   statRcvBuffer[1317] := ' ';
   statRcvBuffer[1318] := ' ';
   statRcvBuffer[1319] := ' ';
   statRcvBuffer[1320] := ' ';
   statRcvBuffer[1321] := ' ';
   statRcvBuffer[1322] := ' ';
   statRcvBuffer[1323] := ' ';
   statRcvBuffer[1324] := ' ';
   statRcvBuffer[1325] := ' ';
   statRcvBuffer[1326] := ' ';
   statRcvBuffer[1327] := ' ';
   statRcvBuffer[1328] := ' ';
   statRcvBuffer[1329] := ' ';
   statRcvBuffer[1330] := ' ';
   statRcvBuffer[1331] := ' ';
   statRcvBuffer[1332] := ' ';
   statRcvBuffer[1333] := ' ';
   statRcvBuffer[1334] := ' ';
   statRcvBuffer[1335] := ' ';
   statRcvBuffer[1336] := ' ';
   statRcvBuffer[1337] := ' ';
   statRcvBuffer[1338] := ' ';
   statRcvBuffer[1339] := ' ';
   statRcvBuffer[1340] := ' ';
   statRcvBuffer[1341] := ' ';
   statRcvBuffer[1342] := ' ';
   statRcvBuffer[1343] := ' ';
   statRcvBuffer[1344] := ' ';
   statRcvBuffer[1345] := ' ';
   statRcvBuffer[1346] := ' ';
   statRcvBuffer[1347] := ' ';
   statRcvBuffer[1348] := ' ';
   statRcvBuffer[1349] := ' ';
   statRcvBuffer[1350] := ' ';
   statRcvBuffer[1351] := ' ';
   statRcvBuffer[1352] := ' ';
   statRcvBuffer[1353] := ' ';
   statRcvBuffer[1354] := ' ';
   statRcvBuffer[1355] := ' ';
   statRcvBuffer[1356] := ' ';
   statRcvBuffer[1357] := ' ';
   statRcvBuffer[1358] := ' ';
   statRcvBuffer[1359] := ' ';
   statRcvBuffer[1360] := ' ';
   statRcvBuffer[1361] := ' ';
   statRcvBuffer[1362] := ' ';
   statRcvBuffer[1363] := ' ';
   statRcvBuffer[1364] := ' ';
   statRcvBuffer[1365] := ' ';
   statRcvBuffer[1366] := ' ';
   statRcvBuffer[1367] := ' ';
   statRcvBuffer[1368] := ' ';
   statRcvBuffer[1369] := ' ';
   statRcvBuffer[1370] := ' ';
   statRcvBuffer[1371] := ' ';
   statRcvBuffer[1372] := ' ';
   statRcvBuffer[1373] := ' ';
   statRcvBuffer[1374] := ' ';
   statRcvBuffer[1375] := ' ';
   statRcvBuffer[1376] := ' ';
   statRcvBuffer[1377] := ' ';
   statRcvBuffer[1378] := ' ';
   statRcvBuffer[1379] := ' ';
   statRcvBuffer[1380] := ' ';
   statRcvBuffer[1381] := ' ';
   statRcvBuffer[1382] := ' ';
   statRcvBuffer[1383] := ' ';
   statRcvBuffer[1384] := ' ';
   statRcvBuffer[1385] := ' ';
   statRcvBuffer[1386] := ' ';
   statRcvBuffer[1387] := ' ';
   statRcvBuffer[1388] := ' ';
   statRcvBuffer[1389] := ' ';
   statRcvBuffer[1390] := ' ';
   statRcvBuffer[1391] := ' ';
   statRcvBuffer[1392] := ' ';
   statRcvBuffer[1393] := ' ';
   statRcvBuffer[1394] := ' ';
   statRcvBuffer[1395] := ' ';
   statRcvBuffer[1396] := ' ';
   statRcvBuffer[1397] := ' ';
   statRcvBuffer[1398] := ' ';
   statRcvBuffer[1399] := ' ';
   statRcvBuffer[1400] := ' ';
   statRcvBuffer[1401] := ' ';
   statRcvBuffer[1402] := ' ';
   statRcvBuffer[1403] := ' ';
   statRcvBuffer[1404] := ' ';
   statRcvBuffer[1405] := ' ';
   statRcvBuffer[1406] := ' ';
   statRcvBuffer[1407] := ' ';
   statRcvBuffer[1408] := ' ';
   statRcvBuffer[1409] := ' ';
   statRcvBuffer[1410] := ' ';
   statRcvBuffer[1411] := ' ';
   statRcvBuffer[1412] := ' ';
   statRcvBuffer[1413] := ' ';
   statRcvBuffer[1414] := ' ';
   statRcvBuffer[1415] := ' ';
   statRcvBuffer[1416] := ' ';
   statRcvBuffer[1417] := ' ';
   statRcvBuffer[1418] := ' ';
   statRcvBuffer[1419] := ' ';
   statRcvBuffer[1420] := ' ';
   statRcvBuffer[1421] := ' ';
   statRcvBuffer[1422] := ' ';
   statRcvBuffer[1423] := ' ';
   statRcvBuffer[1424] := ' ';
   statRcvBuffer[1425] := ' ';
   statRcvBuffer[1426] := ' ';
   statRcvBuffer[1427] := ' ';
   statRcvBuffer[1428] := ' ';
   statRcvBuffer[1429] := ' ';
   statRcvBuffer[1430] := ' ';
   statRcvBuffer[1431] := ' ';
   statRcvBuffer[1432] := ' ';
   statRcvBuffer[1433] := ' ';
   statRcvBuffer[1434] := ' ';
   statRcvBuffer[1435] := ' ';
   statRcvBuffer[1436] := ' ';
   statRcvBuffer[1437] := ' ';
   statRcvBuffer[1438] := ' ';
   statRcvBuffer[1439] := ' ';
   statRcvBuffer[1440] := ' ';
   statRcvBuffer[1441] := ' ';
   statRcvBuffer[1442] := ' ';
   statRcvBuffer[1443] := ' ';
   statRcvBuffer[1444] := ' ';
   statRcvBuffer[1445] := ' ';
   statRcvBuffer[1446] := ' ';
   statRcvBuffer[1447] := ' ';
   statRcvBuffer[1448] := ' ';
   statRcvBuffer[1449] := ' ';
   statRcvBuffer[1450] := ' ';
   statRcvBuffer[1451] := ' ';
   statRcvBuffer[1452] := ' ';
   statRcvBuffer[1453] := ' ';
   statRcvBuffer[1454] := ' ';
   statRcvBuffer[1455] := ' ';
   statRcvBuffer[1456] := ' ';
   statRcvBuffer[1457] := ' ';
   statRcvBuffer[1458] := ' ';
   statRcvBuffer[1459] := ' ';
   statSizeRcvArray := 101;
   statDataIsString := TRUE;
END_DATA_BLOCK

DATA_BLOCK "LHTTP_parameters"   // DB3
{ S7_Optimized_Access := 'TRUE' }
VERSION : 0.1
   VAR
      hwID : Hw_Any := 0;
      connID : Conn_Ouc := 16#0001;
      url : String := '192.168.0.56:55555/resource';
      contentType : String := 'application/json';
      Head : String := 'Authorization: Basic dGVzdDEyMzQ1OnRlc3QxMjM0NQ==$00';
      HeaderData : Array[0..255] of Char;
      responseData : Array[0..100] of Char;
   END_VAR
BEGIN
   responseData[100] := ' ';
   responseData[99] := ' ';
   responseData[98] := ' ';
   responseData[97] := ' ';
   responseData[96] := ' ';
   responseData[95] := ' ';
   responseData[94] := ' ';
   responseData[93] := ' ';
   responseData[92] := ' ';
   responseData[91] := ' ';
   responseData[90] := ' ';
   responseData[89] := ' ';
   responseData[88] := ' ';
   responseData[87] := ' ';
   responseData[86] := ' ';
   responseData[85] := ' ';
   responseData[84] := ' ';
   responseData[83] := ' ';
   responseData[82] := ' ';
   responseData[81] := ' ';
   responseData[80] := ' ';
   responseData[79] := '}';
   responseData[78] := '"';
   responseData[77] := 'e';
   responseData[76] := 'c';
   responseData[75] := 'r';
   responseData[74] := 'u';
   responseData[73] := 'o';
   responseData[72] := 's';
   responseData[71] := 'e';
   responseData[70] := 'r';
   responseData[69] := ' ';
   responseData[68] := 'e';
   responseData[67] := 'l';
   responseData[66] := 'p';
   responseData[65] := 'm';
   responseData[64] := 'a';
   responseData[63] := 'x';
   responseData[62] := 'e';
   responseData[61] := ' ';
   responseData[60] := 'n';
   responseData[59] := 'a';
   responseData[58] := ' ';
   responseData[57] := 's';
   responseData[56] := 'i';
   responseData[55] := ' ';
   responseData[54] := 's';
   responseData[53] := 'i';
   responseData[52] := 'h';
   responseData[51] := 'T';
   responseData[50] := '"';
   responseData[49] := ':';
   responseData[48] := '"';
   responseData[47] := 'n';
   responseData[46] := 'o';
   responseData[45] := 'i';
   responseData[44] := 't';
   responseData[43] := 'p';
   responseData[42] := 'i';
   responseData[41] := 'r';
   responseData[40] := 'c';
   responseData[39] := 's';
   responseData[38] := 'e';
   responseData[37] := 'd';
   responseData[36] := '"';
   responseData[35] := ',';
   responseData[34] := '"';
   responseData[33] := 'e';
   responseData[32] := 'c';
   responseData[31] := 'r';
   responseData[30] := 'u';
   responseData[29] := 'o';
   responseData[28] := 's';
   responseData[27] := 'e';
   responseData[26] := 'r';
   responseData[25] := ' ';
   responseData[24] := 'e';
   responseData[23] := 'l';
   responseData[22] := 'p';
   responseData[21] := 'm';
   responseData[20] := 'a';
   responseData[19] := 'x';
   responseData[18] := 'e';
   responseData[17] := '"';
   responseData[16] := ':';
   responseData[15] := '"';
   responseData[14] := 'e';
   responseData[13] := 'm';
   responseData[12] := 'a';
   responseData[11] := 'n';
   responseData[10] := '"';
   responseData[9] := ',';
   responseData[8] := '"';
   responseData[7] := '1';
   responseData[6] := '"';
   responseData[5] := ':';
   responseData[4] := '"';
   responseData[3] := 'd';
   responseData[2] := 'i';
   responseData[1] := '"';
   responseData[0] := '{';
   HeaderData[0] := 'A';
   HeaderData[1] := 'u';
   HeaderData[2] := 't';
   HeaderData[3] := 'h';
   HeaderData[4] := 'o';
   HeaderData[5] := 'r';
   HeaderData[6] := 'i';
   HeaderData[7] := 'z';
   HeaderData[8] := 'a';
   HeaderData[9] := 't';
   HeaderData[10] := 'i';
   HeaderData[11] := 'o';
   HeaderData[12] := 'n';
   HeaderData[13] := ':';
   HeaderData[14] := ' ';
   HeaderData[15] := 'B';
   HeaderData[16] := 'a';
   HeaderData[17] := 's';
   HeaderData[18] := 'i';
   HeaderData[19] := 'c';
   HeaderData[20] := ' ';
   HeaderData[21] := 'd';
   HeaderData[22] := 'G';
   HeaderData[23] := 'V';
   HeaderData[24] := 'z';
   HeaderData[25] := 'd';
   HeaderData[26] := 'D';
   HeaderData[27] := 'E';
   HeaderData[28] := 'y';
   HeaderData[29] := 'M';
   HeaderData[30] := 'z';
   HeaderData[31] := 'Q';
   HeaderData[32] := '1';
   HeaderData[33] := 'O';
   HeaderData[34] := 'n';
   HeaderData[35] := 'R';
   HeaderData[36] := 'l';
   HeaderData[37] := 'c';
   HeaderData[38] := '3';
   HeaderData[39] := 'Q';
   HeaderData[40] := 'x';
   HeaderData[41] := 'M';
   HeaderData[42] := 'j';
   HeaderData[43] := 'M';
   HeaderData[44] := '0';
   HeaderData[45] := 'N';
   HeaderData[46] := 'Q';
   HeaderData[47] := '=';
   HeaderData[48] := '=';
   HeaderData[49] := '$00';
   HeaderData[50] := ' ';
   HeaderData[51] := ' ';
   HeaderData[52] := ' ';
   HeaderData[53] := ' ';
   HeaderData[54] := ' ';
   HeaderData[55] := ' ';
   HeaderData[56] := ' ';
   HeaderData[57] := ' ';
   HeaderData[58] := ' ';
   HeaderData[59] := ' ';
   HeaderData[60] := ' ';
   HeaderData[61] := ' ';
   HeaderData[62] := ' ';
   HeaderData[63] := ' ';
   HeaderData[64] := ' ';
   HeaderData[65] := ' ';
   HeaderData[66] := ' ';
   HeaderData[67] := ' ';
   HeaderData[68] := ' ';
   HeaderData[69] := ' ';
   HeaderData[70] := ' ';
   HeaderData[71] := ' ';
   HeaderData[72] := ' ';
   HeaderData[73] := ' ';
   HeaderData[74] := ' ';
   HeaderData[75] := ' ';
   HeaderData[76] := ' ';
   HeaderData[77] := ' ';
   HeaderData[78] := ' ';
   HeaderData[79] := ' ';
   HeaderData[80] := ' ';
   HeaderData[81] := ' ';
   HeaderData[82] := ' ';
   HeaderData[83] := ' ';
   HeaderData[84] := ' ';
   HeaderData[85] := ' ';
   HeaderData[86] := ' ';
   HeaderData[87] := ' ';
   HeaderData[88] := ' ';
   HeaderData[89] := ' ';
   HeaderData[90] := ' ';
   HeaderData[91] := ' ';
   HeaderData[92] := ' ';
   HeaderData[93] := ' ';
   HeaderData[94] := ' ';
   HeaderData[95] := ' ';
   HeaderData[96] := ' ';
   HeaderData[97] := ' ';
   HeaderData[98] := ' ';
   HeaderData[99] := ' ';
   HeaderData[100] := ' ';
   HeaderData[101] := ' ';
   HeaderData[102] := ' ';
   HeaderData[103] := ' ';
   HeaderData[104] := ' ';
   HeaderData[105] := ' ';
   HeaderData[106] := ' ';
   HeaderData[107] := ' ';
   HeaderData[108] := ' ';
   HeaderData[109] := ' ';
   HeaderData[110] := ' ';
   HeaderData[111] := ' ';
   HeaderData[112] := ' ';
   HeaderData[113] := ' ';
   HeaderData[114] := ' ';
   HeaderData[115] := ' ';
   HeaderData[116] := ' ';
   HeaderData[117] := ' ';
   HeaderData[118] := ' ';
   HeaderData[119] := ' ';
   HeaderData[120] := ' ';
   HeaderData[121] := ' ';
   HeaderData[122] := ' ';
   HeaderData[123] := ' ';
   HeaderData[124] := ' ';
   HeaderData[125] := ' ';
   HeaderData[126] := ' ';
   HeaderData[127] := ' ';
   HeaderData[128] := ' ';
   HeaderData[129] := ' ';
   HeaderData[130] := ' ';
   HeaderData[131] := ' ';
   HeaderData[132] := ' ';
   HeaderData[133] := ' ';
   HeaderData[134] := ' ';
   HeaderData[135] := ' ';
   HeaderData[136] := ' ';
   HeaderData[137] := ' ';
   HeaderData[138] := ' ';
   HeaderData[139] := ' ';
   HeaderData[140] := ' ';
   HeaderData[141] := ' ';
   HeaderData[142] := ' ';
   HeaderData[143] := ' ';
   HeaderData[144] := ' ';
   HeaderData[145] := ' ';
   HeaderData[146] := ' ';
   HeaderData[147] := ' ';
   HeaderData[148] := ' ';
   HeaderData[149] := ' ';
   HeaderData[150] := ' ';
   HeaderData[151] := ' ';
   HeaderData[152] := ' ';
   HeaderData[153] := ' ';
   HeaderData[154] := ' ';
   HeaderData[155] := ' ';
   HeaderData[156] := ' ';
   HeaderData[157] := ' ';
   HeaderData[158] := ' ';
   HeaderData[159] := ' ';
   HeaderData[160] := ' ';
   HeaderData[161] := ' ';
   HeaderData[162] := ' ';
   HeaderData[163] := ' ';
   HeaderData[164] := ' ';
   HeaderData[165] := ' ';
   HeaderData[166] := ' ';
   HeaderData[167] := ' ';
   HeaderData[168] := ' ';
   HeaderData[169] := ' ';
   HeaderData[170] := ' ';
   HeaderData[171] := ' ';
   HeaderData[172] := ' ';
   HeaderData[173] := ' ';
   HeaderData[174] := ' ';
   HeaderData[175] := ' ';
   HeaderData[176] := ' ';
   HeaderData[177] := ' ';
   HeaderData[178] := ' ';
   HeaderData[179] := ' ';
   HeaderData[180] := ' ';
   HeaderData[181] := ' ';
   HeaderData[182] := ' ';
   HeaderData[183] := ' ';
   HeaderData[184] := ' ';
   HeaderData[185] := ' ';
   HeaderData[186] := ' ';
   HeaderData[187] := ' ';
   HeaderData[188] := ' ';
   HeaderData[189] := ' ';
   HeaderData[190] := ' ';
   HeaderData[191] := ' ';
   HeaderData[192] := ' ';
   HeaderData[193] := ' ';
   HeaderData[194] := ' ';
   HeaderData[195] := ' ';
   HeaderData[196] := ' ';
   HeaderData[197] := ' ';
   HeaderData[198] := ' ';
   HeaderData[199] := ' ';
   HeaderData[200] := ' ';
   HeaderData[201] := ' ';
   HeaderData[202] := ' ';
   HeaderData[203] := ' ';
   HeaderData[204] := ' ';
   HeaderData[205] := ' ';
   HeaderData[206] := ' ';
   HeaderData[207] := ' ';
   HeaderData[208] := ' ';
   HeaderData[209] := ' ';
   HeaderData[210] := ' ';
   HeaderData[211] := ' ';
   HeaderData[212] := ' ';
   HeaderData[213] := ' ';
   HeaderData[214] := ' ';
   HeaderData[215] := ' ';
   HeaderData[216] := ' ';
   HeaderData[217] := ' ';
   HeaderData[218] := ' ';
   HeaderData[219] := ' ';
   HeaderData[220] := ' ';
   HeaderData[221] := ' ';
   HeaderData[222] := ' ';
   HeaderData[223] := ' ';
   HeaderData[224] := ' ';
   HeaderData[225] := ' ';
   HeaderData[226] := ' ';
   HeaderData[227] := ' ';
   HeaderData[228] := ' ';
   HeaderData[229] := ' ';
   HeaderData[230] := ' ';
   HeaderData[231] := ' ';
   HeaderData[232] := ' ';
   HeaderData[233] := ' ';
   HeaderData[234] := ' ';
   HeaderData[235] := ' ';
   HeaderData[236] := ' ';
   HeaderData[237] := ' ';
   HeaderData[238] := ' ';
   HeaderData[239] := ' ';
   HeaderData[240] := ' ';
   HeaderData[241] := ' ';
   HeaderData[242] := ' ';
   HeaderData[243] := ' ';
   HeaderData[244] := ' ';
   HeaderData[245] := ' ';
   HeaderData[246] := ' ';
   HeaderData[247] := ' ';
   HeaderData[248] := ' ';
   HeaderData[249] := ' ';
   HeaderData[250] := ' ';
   HeaderData[251] := ' ';
   HeaderData[252] := ' ';
   HeaderData[253] := ' ';
   HeaderData[254] := ' ';
   HeaderData[255] := ' ';
END_DATA_BLOCK

DATA_BLOCK "LHTTP_control"   // DB5
{ S7_Optimized_Access := 'TRUE' }
VERSION : 0.1
   VAR
      PUT_POST : Bool;
      GET : Bool;
      ExtractedDataName : String;
      ExtractedDataDescription : String;
      ExtractedDataMessage : String;
      RequestPayload : String := '{"id":"1","name":"example resource","description":"This is an example resource"}';
      geturl : String := '192.168.0.56:55555/resource/1';
      PostOrPut : USInt := 0;   // 0=post , 1=put
   END_VAR
BEGIN
END_DATA_BLOCK

// folder: (top level)

ORGANIZATION_BLOCK "Main"   // OB1, LAD, ProgramCycle
TITLE = "Main Program Sweep (Cycle)"
{ S7_Optimized_Access := 'TRUE' }
VERSION : 0.1
   VAR_INPUT
      Initial_Call : Bool;   // Initial call of this OB
      Remanence : Bool;   // =True, if remanent data are available
   END_VAR
BEGIN

REGION Network 1
   // Download password 1234
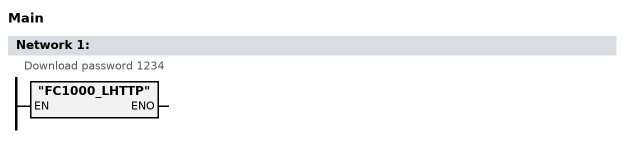
   RUNG wire#powerrail
      "FC1000_LHTTP"()
   END_RUNG
   // the same network as SCL:
   "FC1000_LHTTP"();
END_REGION
END_ORGANIZATION_BLOCK

// folder: 1000_HTTP

FUNCTION "FC1000_LHTTP" : Void   // FC1000, FBD
{ S7_Optimized_Access := 'TRUE' }
VERSION : 0.1
BEGIN

REGION Network 1: Header Data Additions - Convert String to Chars
   // Header fields are separated by an end-ofline ("$R$L"). The end of the user-defined header fields is signaled to the FB with the character 
   // "$00"
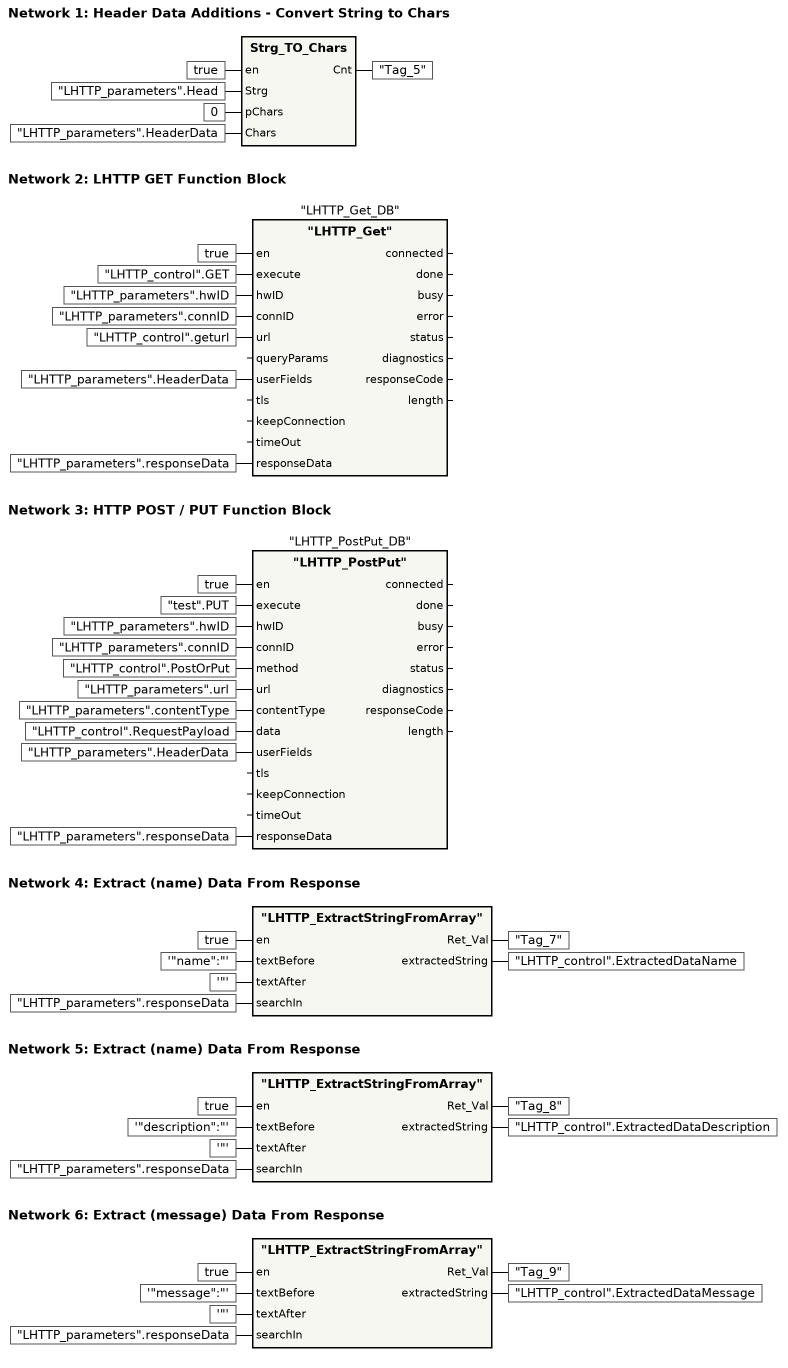
   // no SCL statement known for Strg_TO_Chars: written as a call
   IF true THEN
       Strg_TO_Chars(Strg := "LHTTP_parameters".Head,
                     pChars := 0,
                     Chars := "LHTTP_parameters".HeaderData,
                     Cnt => "Tag_5");
   END_IF;
END_REGION

REGION Network 2: LHTTP GET Function Block
   IF true THEN
       "LHTTP_Get_DB"(execute := "LHTTP_control".GET,   // "LHTTP_Get"
                      hwID := "LHTTP_parameters".hwID,
                      connID := "LHTTP_parameters".connID,
                      url := "LHTTP_control".geturl,
                      userFields := "LHTTP_parameters".HeaderData,
                      responseData := "LHTTP_parameters".responseData);
   END_IF;
END_REGION

REGION Network 3: HTTP POST / PUT Function Block
   IF true THEN
       "LHTTP_PostPut_DB"(execute := "test".PUT,   // "LHTTP_PostPut"
                          hwID := "LHTTP_parameters".hwID,
                          connID := "LHTTP_parameters".connID,
                          method := "LHTTP_control".PostOrPut,
                          url := "LHTTP_parameters".url,
                          contentType := "LHTTP_parameters".contentType,
                          data := "LHTTP_control".RequestPayload,
                          userFields := "LHTTP_parameters".HeaderData,
                          responseData := "LHTTP_parameters".responseData);
   END_IF;
END_REGION

REGION Network 4: Extract (name) Data From Response
   IF true THEN
       "Tag_7" := "LHTTP_ExtractStringFromArray"(textBefore := '"name":"',
                               textAfter := '"',
                               searchIn := "LHTTP_parameters".responseData,
                               extractedString => "LHTTP_control".ExtractedDataName);
   END_IF;
END_REGION

REGION Network 5: Extract (name) Data From Response
   IF true THEN
       "Tag_8" := "LHTTP_ExtractStringFromArray"(textBefore := '"description":"',
                               textAfter := '"',
                               searchIn := "LHTTP_parameters".responseData,
                               extractedString => "LHTTP_control".ExtractedDataDescription);
   END_IF;
END_REGION

REGION Network 6: Extract (message) Data From Response
   IF true THEN
       "Tag_9" := "LHTTP_ExtractStringFromArray"(textBefore := '"message":"',
                               textAfter := '"',
                               searchIn := "LHTTP_parameters".responseData,
                               extractedString => "LHTTP_control".ExtractedDataMessage);
   END_IF;
END_REGION
END_FUNCTION

// folder: 1000_HTTP/LHTTP

FUNCTION_BLOCK "LHTTP_Get"   // FB8, SCL
TITLE = LHTTP_Get
{ S7_Optimized_Access := 'TRUE' }
AUTHOR : Siemens Industry Online Support
FAMILY : LHTTP
VERSION : 2.1
// Implements the HTTP GET method
   VAR_INPUT
      execute : Bool;   // Send HTTP request
      hwID : Hw_Any;   // Hardware ID of Ethernet interface
      connID : Conn_Ouc := 1;   // Unique connection ID
      url : String;   // URL, i.e. "http://www.siemens.com/simatic"
      queryParams : String;   // Additional query parameters if "url" is not long enough, i.e. "lang=en&q=simatic"; "?" or "&" is inserted automatically in between "url" and "queryParameters". / Optional query parameters that are appended to URL, i.e. "lang=en&q=simatic"
      userFields : Array[0..#UPPER_USER_FIELDS] of Char;   // Additional user-defined header fields
      tls : "LHTTP_typeTLS";   // TLS certificates for secure connections (HTTPS), leave open for non-secure connections (HTTP)
      keepConnection : Bool;   // Keep connection established after execution of request
      timeOut : Time := T#10s;   // Time to wait for response from server
   END_VAR
   VAR_OUTPUT
      connected : Bool;   // Connection to web server is established
      done : Bool;   // HTTP request finished
      busy : Bool;   // Function is busy
      error : Bool;   // An error occured
      status : Word := 16#7000;   // Specifies the error
      diagnostics : "typeDiagnostics";   // Diagnostics information of FB
      responseCode : UInt;   // HTTP response code
      length : UDInt;   // Length of received data
   END_VAR
   VAR_IN_OUT
      responseData : Array[*] of Char;   // Data received from HTTP server
   END_VAR
   VAR
      instTSendC : TSEND_C;   // Instance of TSEND_C
      instTRcv : TRCV;   // Instance of TRCV
      instTimeout : TON_TIME;   // Time-out
      statConnected : Bool;   // Static value for output 'connected'
      statDone : Bool;   // Static value for output 'done'
      statBusy : Bool;   // Static value for output 'busy'
      statError : Bool;   // Static value for output 'error'
      statStatus : Word := 16#7000;   // Static value for output 'status'
      statResponseCode : UInt;   // Static value for output 'responseCode'
      statLength : UDInt;   // Static value for output 'length'
      statFBState : USInt := 0;   // Current state in state machine
      statSubfunctionStatus : DWord;   // Status or return value of called FBs, FCs and system blocks
      statEmptyDiagnostics : "typeDiagnostics";   // Empty diagnostics information (for initialization purposes only)
      statParam : Struct   // Connection parameters
         isQDN : Bool;
         paramQDN : TCON_QDN_SEC;   // Connection parameters in form of QDN
         paramIP : TCON_IP_V4_SEC;   // Connection parameters in form of IP address
      END_STRUCT;
      statHost : String;   // Host part of URL
      statRequest : Struct   // GET request
         chars : Array[0..#UPPER_REQUEST_ARRAY] of Char;   // GET request (max. length: url (254) + data (254) + header (94)
         length : UInt;   // Length of GET request
      END_STRUCT;
      statSend : Struct   // Parameters for instruction TSend_C
         connect : Bool;   // Establish and keep connection
         req : Bool;   // Send data
      END_STRUCT;
      statEncoding : String;   // Transfer encoding of response from HTTP server
      statContentLength : UInt;   // Content length as specified in header of response
      statChunkLen : UDInt;   // Remaining length of current chunk
      statRcvdLen : UDInt;   // Sum length of received data
      statTimeoutIn : Bool;   // Timeout
      statRcvBuffer : Array[0..#UPPER_TCP_FRAME] of Char;   // Temporary receive buffer
      statSizeRcvArray : UDInt;   // Size of receive buffer at parameter "responseData"
      statExecuteOld : Bool;   // Last cycle's value of input "execute"
   END_VAR
   VAR_TEMP
      tempUrl : String;   // Copy of URL
      tempQuery : String;   // Query part of URL
      tempIndex : DInt;   // Index for for loops
      tempPos : Int;   // General tag for positions
      tempLen : UInt;   // General tag for lengths
      tempRet : Word;   // General tag for return values
      tempString : String;   // General tag for strings
      tempExitLoop : Bool;   // Condition to exit REPEAT loop around state machine
      tempChunk : Struct   // Temporary tags for chunked encoding
         posData : UInt;   // Start position of data in current packet
         lenData : UInt;   // Length of data in current packet
         exitLoop : Bool;   // Condition to exit loop
      END_STRUCT;
   END_VAR
   VAR CONSTANT
      UPPER_REQUEST_ARRAY : UInt := 1459;   // Upper limit of request array
      UPPER_TCP_FRAME : UInt := 1459;   // Upper limit of a TCP/IP frame
      UPPER_USER_FIELDS : USInt := 255;   // Upper limit of userFields
      PORT_UNSECURE : UInt := 80;   // Port for unsecure HTTP connection
      PORT_SECURE : UInt := 443;   // Port for secure HTTP connection
      POS_RESPONSE_CODE : USInt := 9;   // Position of HTTP response code in response message
      STATUS_DONE : Word := 16#0000;   // Job finished without errors
      STATUS_DISCONNECTED : Word := 16#0003;   // Communication connection closed
      STATUS_IDLE : Word := 16#7000;   // No job
      STATUS_FIRST_CALL : Word := 16#7001;   // First call after incoming new job (rising edge 'execute')
      STATUS_CONNECTING : Word := 16#7002;   // Connection is currently being established
      STATUS_DISCONNECTING : Word := 16#7003;   // Communication connection is being terminated
      STATUS_MONITORING : Word := 16#7004;   // Communication connection has been established and is being monitored. No send job execution active
      STATUS_SENT : Word := 16#7005;   // Request sent, waiting for response
      SUB_STATUS_NO_ERROR : DWord := 16#0000_0000;   // No error occured in subfunction call
      ERR_BOUND_NOT_ZERO : Word := 16#8201;   // Lower bound of receive buffer is not 0
      ERR_INVALID_URL : Word := 16#8202;   // Invalid URL
      ERR_DIFFERENT_HOST : Word := 16#8203;   // Trying to use existing connection with different host
      ERR_END_USER_FIELDS : Word := 16#8206;   // End of user-defined header fields could not be found
      ERR_REQUEST_SIZE : Word := 16#8210;   // Request array is too small for specified parameters
      ERR_RESPONSE_SIZE : Word := 16#8220;   // Receive buffer at parameter "responseData" too small
      ERR_CONN_LOST : Word := 16#8400;   // Offset for lost connection
      ERR_FORWARDING : Word := 16#8403;   // Server responded with forwarding message. Forwarding is not supported, see "diagnostics"
      ERR_WEBSERVER : Word := 16#8404;   // Webserver responded with error code, see "diagnostics"
      ERR_INVALID_HEADER : Word := 16#8405;   // Header of response is invalid
      ERR_TIMEOUT : Word := 16#8408;   // Time-out occurred
      ERR_UNDEFINED_STATE : Word := 16#8600;   // Error due to an undefined state in state machine
      ERR_TSENDC : Word := 16#8601;   // Error: TCON encountered an error, see "diagnostics"
      ERR_TRCV : Word := 16#8603;   // Error: TURCV encountered error, see "diagnostics"
      ERR_MOVE_USER_FIELDS : Word := 16#8612;   // Error in MOVE_BLK_VARIANT to copy user-defined header fields, see "diagnostics"
      ERR_ENCODING_UNKNOWN : Word := 16#8620;   // Transfer encoding of response could not be detected or is unsupported
      ERR_MOVE_IDENTITY : Word := 16#8630;   // Error in MOVE_BLK_VARIANT for transfer encoding 'identity', see "diagnostics"
      ERR_DECODING_FAILED : Word := 16#8640;   // Chunk encoded response could not be decoded
      ERR_MOVE_CHUNKED : Word := 16#8641;   // Error in MOVE_BLK_VARIANT for transfer encoding 'chunked', see "diagnostics"
      TSENDC_STATUS_CONNECTED : Word := 16#0001;   // TSEND_C: Communication connection established
      MOVE_STATUS_SIZE : Word := 16#8483;   // MOVE_BLK_VARIANT: DEST too small
      FB_STATE_NO_PROCESSING : USInt := 0;   // FB state: No processing
      FB_STATE_INIT : USInt := 1;   // FB state: initialization
      FB_STATE_REQUEST : USInt := 2;   // FB state: prepare request
      FB_STATE_SEND : USInt := 3;   // FB state: send request
      FB_STATE_RCV : USInt := 4;   // FB state: receive data
      FB_STATE_MON : USInt := 5;   // FB state: monitoring connection
      CRLF : String := '$R$L';   // Newline control character (carriage return, line feed)
      HEADER_END : String := '$R$L$R$L';   // End of HTTP header (two newline control characters)
      LEN_CRLF : UInt := 2;   // Length of CRLF
   END_VAR
   // statParam.paramIP.ConnPara.ActiveEstablished := true;
   // statParam.paramQDN.ConnPara.ActiveEstablished := true;
BEGIN
   REGION BLOCK INFO HEADER
     //===============================================================================
     // SIEMENS / (c)Copyright 2021
     //-------------------------------------------------------------------------------
     // Title:        LHTTP_Get
     // Function:     Implements the HTTP GET method
     // Library:      LHTTP
     // Author:       Siemens Industry Online Support
     // Tested with:  CPU 1516-3 PN/DP V2.9
     // Engineering:  TIA Portal V17
     // Restrictions: --
     // Requirements: S7-1200 with firmware V4.4 or higher
     //               S7-1500 with firmware V2.0 or higher
     //-------------------------------------------------------------------------------
     // Change log table:
     // Version  | Date       | Expert in charge       | Changes applied
     //----------|------------|------------------------|------------------------------
     // 02.01.00 | 2021-12-15 | Online Support         | Renamed parameter "data" to "queryParams"
     //-------------------------------------------------------------------------------
     // 02.00.04 | 2021-05-10 | Online Support         | Fixed issues with chunked encoding
     //          |            |                        | Allow chunk sizes > 65535 Bytes
     //          |            |                        | Made header evaluation case-insensitive
     //-------------------------------------------------------------------------------
     // 02.00.00 | 2020-12-16 | Online Support         | Added option to keep connection established
     //          |            |                        | Added parameter to add user-defined headers fields
     //          |            |                        | Changed to data type of "data" to Variant to allow larger data
     //          |            |                        | Removed "statusID" and added "diagnostics" instead, changed some error codes
     //-------------------------------------------------------------------------------
     // 01.00.00 | 2019-04-01 | Online Support         | First released version
     //===============================================================================
   END_REGION

   REGION INSTRUCTIONS
     IF (#statStatus <> #STATUS_IDLE) THEN // Only execute when FB is triggered to reduce system load
       // Connect and send
       IF #statParam.isQDN THEN // Call if host is a domain name
         #instTSendC(REQ     := #statSend.req,
                     CONT    := #statSend.connect,
                     LEN     := #statRequest.length,
                     CONNECT := #statParam.paramQDN,
                     DATA    := #statRequest.chars);
       ELSE // Call if host is an IP address
         #instTSendC(REQ     := #statSend.req,
                     CONT    := #statSend.connect,
                     LEN     := #statRequest.length,
                     CONNECT := #statParam.paramIP,
                     DATA    := #statRequest.chars);
       END_IF;

       // Receive
       #instTRcv(ID    := #statParam.paramQDN.ConnPara.ID,
                 EN_R  := #statFBState >= #FB_STATE_RCV,
                 LEN   := 0,
                 ADHOC := true,
                 DATA  := #statRcvBuffer);

       // Monitor time out
       #instTimeout(IN := #statTimeoutIn,
                    PT := #timeOut);

       IF #instTimeout.Q THEN
         #statStatus := #ERR_TIMEOUT;
       END_IF;
     END_IF;
   END_REGION

   REGION TRIGGERING
     IF (#execute = true AND #statExecuteOld = false) // Check if FB is triggered
       AND (#statStatus = #STATUS_IDLE OR #statStatus = #STATUS_MONITORING)
     THEN // First call; initialize FB
       // Copy URL
       #tempUrl := #url;

       #statBusy := true;
       #statStatus := #STATUS_FIRST_CALL;
       #statSubfunctionStatus := #SUB_STATUS_NO_ERROR;
       #diagnostics := #statEmptyDiagnostics;

       IF #statConnected = FALSE THEN // Connection is not yet established
         #statFBState := #FB_STATE_INIT;
       ELSE // Connection is already established, skip init
         #statFBState := #FB_STATE_REQUEST;
       END_IF;

     ELSIF (#statStatus = #STATUS_FIRST_CALL) THEN
       #statStatus := #STATUS_CONNECTING;
     END_IF;

     // Edge detection 'execute' input
     #statExecuteOld := #execute;
   END_REGION TRIGGERING

   IF (#statStatus = #STATUS_IDLE) THEN // Nothing to do -> End here to reduce "system load"
     RETURN;
   END_IF;

   REGION STATE_MACHINE
     // State machine is wrapped in REPEAT loop to make it possible to quickly exit state machine
     // in case of an error or to go through CASE multiple times within one cycle
     REPEAT
       #tempExitLoop := true; // Condition to exit loop is set per default

       CASE #statFBState OF // State machine of FB
         #FB_STATE_NO_PROCESSING: // No processing active
           ;

         #FB_STATE_INIT:
           REGION INIT
             // Get size of receive buffer
             IF LOWER_BOUND(ARR := #responseData, DIM := 1) <> 0 THEN
               #statStatus := #ERR_BOUND_NOT_ZERO;
               EXIT;
             ELSE
               #statSizeRcvArray := DINT_TO_UDINT(UPPER_BOUND(ARR := #responseData, DIM := 1)) + 1;
             END_IF;

             // Set connection parameters
             #statParam.paramQDN.ConnPara.InterfaceId := #hwID;
             #statParam.paramQDN.ConnPara.ID := #connID;
             #statParam.paramIP.ConnPara.InterfaceId := #hwID;
             #statParam.paramIP.ConnPara.ID := #connID;

             // Check if network protocol was specified to determine if connection should be secured
             #tempPos := FIND(IN1 := #tempUrl, IN2 := 'https://');
             IF #tempPos = 1 THEN // HTTPS
               #statParam.paramQDN.ActivateSecureConn := true;
               #statParam.paramQDN.ExtTLSCapabilities.%X0 := #tls.validateServerIdentity;
               #statParam.paramQDN.TLSServerCertRef := #tls.serverCert;
               #statParam.paramQDN.TLSClientCertRef := #tls.clientCert;
               #statParam.paramIP.ActivateSecureConn := true;
               #statParam.paramIP.ExtTLSCapabilities.%X0 := #tls.validateServerIdentity;
               #statParam.paramIP.TLSServerCertRef := #tls.serverCert;
               #statParam.paramIP.TLSClientCertRef := #tls.clientCert;
               // Delete network protocol from URL
               #tempUrl := DELETE(IN := #tempUrl, L := 8, P := 1);
             ELSE // HTTP
               #statParam.paramQDN.ActivateSecureConn := false;
               #statParam.paramIP.ActivateSecureConn := false;
               // Delete network protocol from URL if specified
               IF #tempUrl[5] = ':' THEN
                 #tempUrl := DELETE(IN := #tempUrl, L := 7, P := 1);
               END_IF;
             END_IF;

             // Determine if host is domain name or IP address
             #tempPos := CHAR_TO_INT(#tempUrl[1]);
             IF #tempPos >= CHAR_TO_INT('A') AND #tempPos <= CHAR_TO_INT('z') THEN // Host is a domain name
               #statParam.isQDN := true;
             ELSIF #tempPos >= CHAR_TO_INT('0') AND #tempPos <= CHAR_TO_INT('9') THEN // Host is an IP address
               #statParam.isQDN := false;
             ELSE // URL invalid
               #statStatus := #ERR_INVALID_URL;
               EXIT;
             END_IF;

             // Get host name and port
             #tempPos := FIND(IN1 := #tempUrl, IN2 := '/');
             IF #tempPos > 0 THEN // URL has a path after host name
               #statHost := LEFT(IN := #tempUrl, L := #tempPos - 1);
             ELSE
               #statHost := #tempUrl;
             END_IF;
             #tempPos := FIND(IN1 := #statHost, IN2 := ':');
             IF #tempPos > 0 THEN // Port specified in URL
               #statParam.paramQDN.ConnPara.RemotePort := STRING_TO_UINT(DELETE(IN := #statHost, L := #tempPos, P := 1));
               #statParam.paramIP.ConnPara.RemotePort := STRING_TO_UINT(DELETE(IN := #statHost, L := #tempPos, P := 1));
               #statHost := LEFT(IN := #statHost, L := #tempPos - 1);
             ELSE // No port specified in URL, set default port
               IF #statParam.paramQDN.ActivateSecureConn OR #statParam.paramIP.ActivateSecureConn THEN
                 #statParam.paramQDN.ConnPara.RemotePort := #PORT_SECURE;
                 #statParam.paramIP.ConnPara.RemotePort := #PORT_SECURE;
               ELSE
                 #statParam.paramQDN.ConnPara.RemotePort := #PORT_UNSECURE;
                 #statParam.paramIP.ConnPara.RemotePort := #PORT_UNSECURE;
               END_IF;
             END_IF;

             IF #statParam.isQDN THEN // Host is a domain name
               #statParam.paramQDN.ConnPara.RemoteQDN := CONCAT(IN1 := #statHost, IN2 := '.');
             ELSE // Host is an IP address
               #tempString := #statHost;
               FOR #tempIndex := 1 TO 3 DO
                 #tempPos := FIND(IN1 := #tempString, IN2 := '.');
                 #statParam.paramIP.ConnPara.RemoteAddress.ADDR[#tempIndex] := UINT_TO_BYTE(STRING_TO_UINT(LEFT(IN := #tempString, L := #tempPos - 1)));
                 #tempString := DELETE(IN := #tempString, L := #tempPos, P := 1);
               END_FOR;
               #statParam.paramIP.ConnPara.RemoteAddress.ADDR[4] := UINT_TO_BYTE(STRING_TO_UINT(#tempString));
             END_IF;

             #statFBState := #FB_STATE_REQUEST;
             #tempExitLoop := FALSE; // Don't exit loop to go directly to prepare request
           END_REGION INIT

         #FB_STATE_REQUEST:
           REGION PREP_REQUEST
             // Check host in URL when using existing connection
             IF #statConnected = TRUE THEN
               #tempPos := FIND(IN1 := #tempUrl, IN2 := #statHost);
               IF #tempPos = 0 THEN // URL doesn't contain expected host
                 #statStatus := #ERR_DIFFERENT_HOST;
                 EXIT;
               ELSE // Scheme and host must be deleted for further processing
                 #tempUrl := DELETE(IN := #tempUrl, L := #tempPos + LEN(#statHost) - 1, P := 1);
               END_IF;
             END_IF;

             // Get path
             #tempPos := FIND(IN1 := #tempUrl, IN2 := '/');
             IF #tempPos > 0 THEN // URL has a path after host name
               #tempString := DELETE(IN := #tempUrl, L := #tempPos - 1, P := 1);
             ELSE
               #tempString := '/';
             END_IF;

             // Prepare query part of URL
             IF #queryParams <> '' THEN // Parameter is in use
               IF #queryParams[1] = '?' OR #queryParams[1] = '&' THEN
                 #tempQuery := DELETE(IN := #queryParams, P := 1, L := 1);
               ELSE
                 #tempQuery := #queryParams;
               END_IF;
               #tempPos := FIND(IN1 := #tempString, IN2 := '?'); // Check if URL already contains query parameters
               IF #tempPos <> 0 THEN // URL already contains query parameters
                 #tempQuery := CONCAT(IN1 := '&', IN2 := #tempQuery); // Append query parameters with &
               ELSE // URL does not contain query parameters
                 #tempQuery := CONCAT(IN1 := '?', IN2 := #tempQuery); // Append query parameters with ?
               END_IF;
             END_IF;

             // Put together GET request
             // Strg_TO_Chars conversion is done several times to utilize maximum length of parameters url and query parameters
             Strg_TO_Chars(Strg   := CONCAT(IN1 := 'GET ', IN2 := #tempString), // Path cannot be longer than 249 characters --> save to use CONCAT
                           pChars := 0,
                           Cnt    => #tempLen,
                           Chars  := #statRequest.chars);
             #tempPos := UINT_TO_INT(#tempLen);

             Strg_TO_Chars(Strg   := #tempQuery,
                           pChars := #tempPos,
                           Cnt    => #tempLen,
                           Chars  := #statRequest.chars);
             #tempPos += UINT_TO_INT(#tempLen);

             Strg_TO_Chars(Strg   := CONCAT(IN1 := ' HTTP/1.1$R$LHost: ', IN2 := #statHost), // Host will not use all 254 characters --> save to use CONCAT
                           pChars := #tempPos,
                           Cnt    => #tempLen,
                           Chars  := #statRequest.chars);
             #tempPos += UINT_TO_INT(#tempLen);

             Strg_TO_Chars(Strg   := '$R$LUser-Agent: SIMATIC Controller (LHTTP)$R$LAccept: text/html$R$LAccept-Encoding: identity$R$LAccept-Charset: utf-8$R$L',
                           pChars := #tempPos,
                           Cnt    => #tempLen,
                           Chars  := #statRequest.chars);
             #tempPos += UINT_TO_INT(#tempLen);

             // Insert additional user-defined header fields
             IF #userFields[0] <> ' ' THEN
               FOR #tempLen := 0 TO #UPPER_USER_FIELDS DO
                 IF #userFields[#tempLen] = '$00' THEN
                   EXIT;
                 END_IF;
               END_FOR;

               IF #tempLen > #UPPER_USER_FIELDS THEN // End not found
                 #statStatus := #ERR_END_USER_FIELDS;
                 EXIT;
               END_IF;

               #tempRet := INT_TO_WORD(MOVE_BLK_VARIANT(SRC := #userFields, COUNT := #tempLen, SRC_INDEX := 0, DEST_INDEX := #tempPos, DEST => #statRequest.chars));

               IF #tempRet = #MOVE_STATUS_SIZE THEN
                 #statStatus := #ERR_REQUEST_SIZE;
                 EXIT;
               ELSIF #tempRet <> 16#0000 THEN
                 #statStatus := #ERR_MOVE_USER_FIELDS;
                 #statSubfunctionStatus := #tempRet;
                 EXIT;
               END_IF;

               #tempPos += UINT_TO_INT(#tempLen);

               // Append CRLF if needed
               IF #statRequest.chars[#tempPos - 2] <> '$R' AND #statRequest.chars[#tempPos - 1] <> '$L' THEN
                 #statRequest.chars[#tempPos] := '$R';
                 #statRequest.chars[#tempPos + 1] := '$L';
                 #tempPos += 2;
               END_IF;
             END_IF;

             // Append end of header section
             Strg_TO_Chars(Strg   := #CRLF,
                           pChars := #tempPos,
                           Cnt    => #tempLen,
                           Chars  := #statRequest.chars);
             #tempPos += UINT_TO_INT(#tempLen);

             // Calculate total length of request
             #statRequest.length := INT_TO_UINT(#tempPos);

             #statSend.connect := true; // Connect
             #statSend.req := true; // Send request
             #statTimeoutIn := true; // Start timer
             #statFBState := #FB_STATE_SEND;
           END_REGION

         #FB_STATE_SEND: // Send data
           REGION SEND
             IF #instTSendC.STATUS = #TSENDC_STATUS_CONNECTED THEN
               #statConnected := TRUE;
             ELSIF #instTSendC.DONE THEN
               #statStatus := #STATUS_SENT;
               #statFBState := #FB_STATE_RCV;
               // Don't exit loop to go directly to receive state
               // without waiting for next cycle so that no responses can be missed
               #tempExitLoop := false;
             ELSIF #instTSendC.ERROR THEN
               #statStatus := #ERR_TSENDC;
               #statSubfunctionStatus := #instTSendC.STATUS;
             END_IF;
           END_REGION

         #FB_STATE_RCV: // Wait for new data
           REGION RCV
             IF #instTRcv.NDR THEN

               REGION HEADER_EVAL
                 // Evaluate header if received packet is first packet
                 IF #statEncoding = '' THEN
                   // Get response code
                   Chars_TO_Strg(Chars  := #statRcvBuffer,
                                 pChars := #POS_RESPONSE_CODE,
                                 Cnt    := 3,
                                 Strg   => #tempString);
                   #statResponseCode := STRING_TO_UINT(#tempString);

                   // Exit loop immediately and output errror if response code shows errors or forwarding
                   IF #statResponseCode >= 300 THEN
                     #tempRet := ATH(IN := #tempString, N := 3, OUT => #statSubfunctionStatus); // Interpret response code as hexadecimal
                     #statSubfunctionStatus := SHR(IN := #statSubfunctionStatus, N := 20);
                     IF #statResponseCode >= 400 THEN
                       #statStatus := #ERR_WEBSERVER;
                     ELSE
                       #statStatus := #ERR_FORWARDING;
                     END_IF;
                     EXIT;
                   END_IF;

                   // Get length of HTTP header
                   #tempLen := DINT_TO_UINT("LHTTP_FindStringInArray"(searchFor := #HEADER_END, searchIn := #statRcvBuffer) + LEN(#HEADER_END));

                   // Exit loop immediately and output errror if header end cannot be found
                   IF #tempLen = 0 THEN
                     #statStatus := #ERR_INVALID_HEADER;
                     EXIT;
                   END_IF;

                   // Search header for content length
                   #tempRet := "LHTTP_ExtractStringFromArray"(textBefore := 'Content-Length: ',
                                                              textAfter := #CRLF,
                                                              extractedString => #tempString,
                                                              searchIn := #statRcvBuffer);

                   IF #tempRet <> 0 THEN // Content length not found; try lower-case
                     #tempRet := "LHTTP_ExtractStringFromArray"(textBefore := 'content-length: ',
                                                                textAfter := #CRLF,
                                                                extractedString => #tempString,
                                                                searchIn := #statRcvBuffer);
                   END_IF;

                   IF #tempRet = 0 THEN // Content length found
                     #statContentLength := STRING_TO_UINT(#tempString);
                     #statEncoding := 'identity';
                   ELSE // Can't detect content length, check if transfer encoding is 'chunked'
                     #tempPos := DINT_TO_INT("LHTTP_FindStringInArray"(searchFor := 'chunked', searchIn := #statRcvBuffer));

                     IF #tempPos >= 0 THEN
                       #statEncoding := 'chunked';
                     ELSE // Exit loop immediately and output error if content length nor transfer encoding can be detected
                       #statStatus := #ERR_ENCODING_UNKNOWN;
                       EXIT;
                     END_IF;
                   END_IF;

                   IF #instTRcv.RCVD_LEN = #tempLen THEN // Packet contains no body, wait for next packet
                     EXIT;
                   END_IF;
                 END_IF;
               END_REGION

               REGION TE_IDENTITY
                 IF #statEncoding = 'identity' THEN // Transfer encoding is 'identity'
                   // Move data from buffer to output; tempLen contains header length during first packet, otherwise 0
                   #tempRet := INT_TO_WORD(MOVE_BLK_VARIANT(SRC := #statRcvBuffer,
                                                                                    COUNT := MIN(IN1 := #instTRcv.RCVD_LEN - #tempLen, IN2 := #statSizeRcvArray - #statRcvdLen), // Move as much as possible to output
                                                                                    SRC_INDEX := #tempLen,
                                                                                    DEST_INDEX := UDINT_TO_DINT(#statRcvdLen),
                                                                                    DEST => #responseData));

                   // Exit loop immediately and output error if data could not be moved
                   IF #tempRet <> 0 THEN
                     #statStatus := #ERR_MOVE_IDENTITY;
                     #statSubfunctionStatus := #tempRet;
                     EXIT;
                   END_IF;

                   // Add length of received packet to sum; tempLen contains header length during first packet, otherwise 0
                   #statRcvdLen += #instTRcv.RCVD_LEN - #tempLen;

                   IF #statRcvdLen > #statSizeRcvArray THEN // Receive buffer too small
                     #statStatus := #ERR_RESPONSE_SIZE;
                     #statLength := #statContentLength; // Output required size of buffer
                   ELSIF #statRcvdLen >= #statContentLength THEN // Everything was received
                     #statStatus := #STATUS_DONE;
                     #statLength := #statRcvdLen;
                   END_IF;
                 END_IF;
               END_REGION

               REGION TE_CHUNKED
                 IF #statEncoding = 'chunked' THEN // Transfer encoding is 'chunked'

                   // Set position of chunk data
                   #tempChunk.posData := #tempLen; // tempLen contains header length during first packet, otherwise 0

                   REPEAT
                     #tempChunk.exitLoop := true; // Condition to exit loop is set per default

                     // Read length of chunk if received packet is first packet or a previous chunk was received completely
                     IF #statChunkLen = 0 THEN
                       // Extract hexadecimal chunk-size field
                       Chars_TO_Strg(Chars  := #statRcvBuffer,
                                     pChars := #tempChunk.posData,
                                     Cnt    := 0,
                                     Strg   => #tempString);
                       #tempPos := FIND(IN1 := #tempString, IN2 := #CRLF);
                       #tempRet := ATH(IN := #tempString, N := #tempPos - 1, OUT => #statChunkLen);
                       // Shift bits to the right depending on length of chunk size, since ATH is left aligned
                       #statChunkLen := SHR(IN := #statChunkLen, N := 4 * INT_TO_UINT(8 - (#tempPos - 1)));

                       // Move start position of data behind chunk-size field
                       #tempChunk.posData += INT_TO_UINT(#tempPos) + 1;

                       // Exit loop immediately and output error if chunk size cannot be detected
                       IF #tempRet <> 0 THEN
                         #statStatus := #ERR_DECODING_FAILED;
                         EXIT;
                       END_IF;
                     END_IF;

                     IF #statChunkLen = 0 THEN // Length was evaluated, chunk contains no data --> final chunk received
                       #statStatus := #STATUS_DONE;
                       #statLength := #statRcvdLen;
                     ELSE // Chunk contains data
                       // Evaluate length of received packet and set length of data accordingly
                       IF #instTRcv.RCVD_LEN = #tempChunk.posData + #statChunkLen + #LEN_CRLF THEN // Chunk was received entirely and packet contains no further chunks
                         #tempChunk.lenData := UDINT_TO_UINT(#statChunkLen); // Output remaining length of chunk
                       ELSIF #instTRcv.RCVD_LEN < #tempChunk.posData + #statChunkLen + #LEN_CRLF THEN // Packet only contains part of chunk
                         #tempChunk.lenData := UDINT_TO_UINT(#instTRcv.RCVD_LEN) - #tempChunk.posData; // Output entire packet without possible chunk-size field
                       ELSIF #instTRcv.RCVD_LEN > #tempChunk.posData + #statChunkLen + #LEN_CRLF THEN // Current packet contains more than one chunk
                         #tempChunk.lenData := UDINT_TO_UINT(#statChunkLen); // Output remaining length of chunk
                         #tempChunk.exitLoop := false; // Execute loop again since packet contains more data
                       ELSE // Can't decode message
                         #statStatus := #ERR_DECODING_FAILED;
                         EXIT;
                       END_IF;

                       // Move received data to output
                       #tempRet := INT_TO_WORD(MOVE_BLK_VARIANT(SRC := #statRcvBuffer,
                                                                                        COUNT := MIN(IN1 := #tempChunk.lenData, IN2 := #statSizeRcvArray - #statRcvdLen), // Move as much as possible to output
                                                                                        SRC_INDEX := #tempChunk.posData,
                                                                                        DEST_INDEX := UDINT_TO_DINT(#statRcvdLen),
                                                                                        DEST => #responseData));

                       // Exit loop immediately and output error if data could not be moved
                       IF #tempRet <> 0 THEN
                         #statStatus := #ERR_MOVE_CHUNKED;
                         #statSubfunctionStatus := #tempRet;
                         EXIT;
                       END_IF;

                       // Move start position of data behind data of current chunk in case packet contains more data; only relevant if REPEAT loop is executed again
                       #tempChunk.posData += #tempChunk.lenData + #LEN_CRLF;

                       // Subtract length of data in current packet from remaining length of chunk and add to sum of received data
                       #statChunkLen -= #tempChunk.lenData;
                       #statRcvdLen += #tempChunk.lenData;

                       IF #statRcvdLen > #statSizeRcvArray THEN // Receive buffer too small
                         #statStatus := #ERR_RESPONSE_SIZE;
                         #statLength := #statRcvdLen; // Output required size of buffer according to so far received chunked messages
                         EXIT;
                       END_IF;
                     END_IF;
                   UNTIL (#tempChunk.exitLoop = true) END_REPEAT;
                 END_IF;
               END_REGION

             ELSIF #instTRcv.ERROR THEN
               #statStatus := #ERR_TRCV;
               #statSubfunctionStatus := #instTRcv.STATUS;
             END_IF;
           END_REGION

         #FB_STATE_MON:
           REGION MONITORING
             IF #keepConnection = FALSE THEN // Trigger to disconnect
               #statSend.connect := FALSE;
               #statDone := FALSE;
               #statBusy := TRUE;
               #statStatus := #STATUS_DISCONNECTING;
             END_IF;

             IF #instTSendC.STATUS = #STATUS_DISCONNECTED THEN
               #statConnected := FALSE;
               #statStatus := #STATUS_DISCONNECTED;
             ELSIF #instTRcv.ERROR THEN
               #statConnected := FALSE;
               #statStatus := #ERR_CONN_LOST OR (#instTRcv.STATUS AND 16#00FF);
             END_IF;
           END_REGION

         ELSE // Undefined state in state machine reached
           #statStatus := #ERR_UNDEFINED_STATE;
       END_CASE;

     UNTIL (#tempExitLoop = true) END_REPEAT;
   END_REGION

   REGION OUTPUTS
     // Write outputs
     IF (#statStatus = #STATUS_DONE) AND (#statDone = false) THEN // Execution finished without errors
       #statDone := true;
       #statBusy := false;
       #statError := false;
       #statSend.connect := #keepConnection;
       #statSend.req := false;
       #statTimeoutIn := false;

       IF #keepConnection THEN
         // execution finished but connection is kept alive --> set state monitoring
         #statFBState := #FB_STATE_MON;
       ELSE
         #statConnected := FALSE;
         // execution finished --> set state no processing
         #statFBState := #FB_STATE_NO_PROCESSING;
       END_IF;

     ELSIF (#statStatus = #STATUS_DISCONNECTED) AND (#statBusy = true) THEN // Connection was terminated separately of send job
       #statConnected := FALSE;
       #statBusy := FALSE;
       // execution finished --> set state no processing
       #statFBState := #FB_STATE_NO_PROCESSING;

     ELSIF (#statStatus.%X15 = true) AND (#statError = false) THEN // Error occurred (#statStatus is 16#8000 to 16#FFFF)
       #statConnected := false;
       #statDone := false;
       #statBusy := false;
       #statError := true;
       #statSend.connect := false; // After error, connection is always terminated
       #statSend.req := false;
       #statTimeoutIn := false;
       // Write diagnostics
       #diagnostics.status := #statStatus;
       #diagnostics.subfunctionStatus := #statSubfunctionStatus;
       #diagnostics.stateNumber := #statFBState;
       // execution aborted --> set state no processing
       #statFBState := #FB_STATE_NO_PROCESSING;

     ELSIF ((#execute = false) AND ((#statDone = true) OR (#statError = true)))
       OR ((#statStatus = #STATUS_DISCONNECTED) AND (#statBusy = false)) // Connection was terminated separately of send job
     THEN // Reset outputs
       #statDone := false;
       #statBusy := false;
       #statError := false;
       #statResponseCode := 0;
       #statLength := 0;
       #statContentLength := 0;
       #statChunkLen := 0;
       #statEncoding := '';
       #statRcvdLen := 0;

       IF #statConnected THEN
         #statStatus := #STATUS_MONITORING;
       ELSE
         #statStatus := #STATUS_IDLE;
       END_IF;
     END_IF;

     // Write static values to outputs
     #connected := #statConnected;
     #done := #statDone;
     #busy := #statBusy;
     #error := #statError;
     #status := #statStatus;
     #responseCode := #statResponseCode;
     #length := #statLength;
     ENO := NOT #statError;
   END_REGION OUTPUTS
END_FUNCTION_BLOCK

FUNCTION_BLOCK "LHTTP_PostPut"   // FB10, SCL
TITLE = LHTTP_PostPut
{ S7_Optimized_Access := 'TRUE' }
AUTHOR : Siemens Industry Online Support
FAMILY : LHTTP
VERSION : 2.1
// Implements the HTTP POST and PUT methods
   VAR_INPUT
      execute : Bool;   // Send HTTP request
      hwID : Hw_Any;   // Hardware ID of Ethernet interface
      connID : Conn_Ouc := 1;   // Unique connection ID
      method : USInt;   // HTTP method; 0: POST, 1: PUT
      url : String;   // URL, i.e. "www.siemens.com/simatic"
      contentType : String := 'text/plain';   // Cotent type of data, i.e. "text/plain"
      data : Variant;   // Data to transmit with request; data type may be String or Array of Char
      userFields : Array[0..#UPPER_USER_FIELDS] of Char;   // Additional user-defined header fields
      tls : "LHTTP_typeTLS";   // TLS certificates for secure connections (HTTPS), leave open for non-secure connections (HTTP)
      keepConnection : Bool;   // Keep connection established after execution of request
      timeOut : Time := T#10s;   // Time to wait for response from server
   END_VAR
   VAR_OUTPUT
      connected : Bool;   // Connection to web server is established
      done : Bool;   // Request was executed successfully
      busy : Bool;   // Function is busy
      error : Bool;   // An error occured
      status : Word := 16#7000;   // Specifies the error
      diagnostics : "typeDiagnostics";   // Diagnostics information of FB
      responseCode : UInt;   // HTTP response code
      length : UDInt;   // Length of received data
   END_VAR
   VAR_IN_OUT
      responseData : Array[*] of Char;   // Data received from HTTP server
   END_VAR
   VAR
      instTSendC : TSEND_C;   // Instance of TSEND_C
      instTRcv : TRCV;   // Instance of TRCV
      instTimeout : TON_TIME;   // Time-out
      statConnected : Bool;   // Static value for output 'connected'
      statDone : Bool;   // Static value for output 'done'
      statBusy : Bool;   // Static value for output 'busy'
      statError : Bool;   // Static value for output 'error'
      statStatus : Word := 16#7000;   // Static value for output 'status'
      statResponseCode : UInt;   // Static value for output 'responseCode'
      statLength : UDInt;   // Static value for output 'length'
      statFBState : USInt := 0;   // Current state in state machine
      statSubfunctionStatus : DWord;   // Status or return value of called FBs, FCs and system blocks
      statEmptyDiagnostics : "typeDiagnostics";   // Empty diagnostics information (for initialization purposes only)
      statParam : Struct   // Connection parameters
         isQDN : Bool;
         paramQDN : TCON_QDN_SEC;   // Connection parameters in form of QDN
         paramIP : TCON_IP_V4_SEC;   // Connection parameters in form of IP address
      END_STRUCT;
      statHost : String;   // Host part of URL
      statRequest : Struct   // POST request
         chars : Array[0..#UPPER_REQUEST_ARRAY] of Char;   // POST request
         length : UInt;   // Length of POST request
      END_STRUCT;
      statSend : Struct   // Parameters for instruction TSEND_C
         connect : Bool;   // Establish and keep connection
         req : Bool;   // Send data
      END_STRUCT;
      statEncoding : String;   // Transfer encoding of response from HTTP server
      statContentLength : UInt;   // Content length as specified in header of response
      statChunkLen : UDInt;   // Remaining length of current chunk
      statRcvdLen : UDInt;   // Sum length f received packet
      statTimeoutIn : Bool;   // Start timer
      statRcvBuffer : Array[0..#UPPER_TCP_FRAME] of Char;   // Temporary receive buffer; maximum segment size for TCP/IP is 1460
      statSizeRcvArray : UDInt;   // Size of receive buffer at parameter "responseData"
      statExecuteOld : Bool;   // Last cycle's value of input "execute"
      statDataIsString : Bool;   // Data type of "data" is String
   END_VAR
   VAR_TEMP
      tempUrl : String;   // Copy of URL
      tempPath : String;   // Path of URL
      tempData : String;   // Copy of data
      tempLenData : UInt;   // Length of data
      tempIndex : DInt;   // General index for loops
      tempPos : Int;   // General tag for positions
      tempLen : UInt;   // General tag for lengths
      tempRet : Word;   // General tag for return values
      tempString : String;   // General tag for strings
      tempExitLoop : Bool;   // Condition to exit REPEAT loop around state machine
      tempChunk : Struct   // Temporary tags for chunked encoding
         posData : UInt;   // Start position of data in current packet
         lenData : UInt;   // Length of data in current packet
         exitLoop : Bool;   // Condition to exit loop
      END_STRUCT;
   END_VAR
   VAR CONSTANT
      METHOD_POST : USInt := 0;   // Method POST
      METHOD_PUT : USInt := 1;   // Method PUT
      UPPER_REQUEST_ARRAY : UInt := 1459;   // Upper limit of request array
      UPPER_TCP_FRAME : UInt := 1459;   // Upper limit of a TCP/IP frame
      UPPER_USER_FIELDS : USInt := 255;   // Upper limit of userFields
      PORT_UNSECURE : UInt := 80;   // Port for unsecure HTTP connection
      PORT_SECURE : UInt := 443;   // Port for secure HTTP connection
      POS_RESPONSE_CODE : USInt := 9;   // Position of HTTP response code in response message
      STATUS_DONE : Word := 16#0000;   // Job finished without errors
      STATUS_DISCONNECTED : Word := 16#0003;   // Communication connection closed
      STATUS_IDLE : Word := 16#7000;   // No job
      STATUS_FIRST_CALL : Word := 16#7001;   // First call after incoming new job (rising edge 'execute')
      STATUS_CONNECTING : Word := 16#7002;   // Intermediate call after job was started
      STATUS_DISCONNECTING : Word := 16#7003;   // Communication connection is being terminated
      STATUS_MONITORING : Word := 16#7004;   // Communication connection has been established and is being monitored. No send job execution active
      STATUS_SENT : Word := 16#7005;   // Request sent, waiting for response
      SUB_STATUS_NO_ERROR : DWord := 16#0000_0000;   // No error occured in subfunction call
      ERR_BOUND_NOT_ZERO : Word := 16#8201;   // Status: Lower bound of receive buffer is not 0
      ERR_INVALID_URL : Word := 16#8202;   // Status: Invalid URL
      ERR_DIFFERENT_HOST : Word := 16#8203;   // Trying to use existing connection with different host
      ERR_TYPE_DATA : Word := 16#8204;   // Data type of "data" is neither String nor Array of Char
      ERR_END_DATA : Word := 16#8205;   // End of data could not be found
      ERR_END_USER_FIELDS : Word := 16#8206;   // End of user-defined header fields could not be found
      ERR_METHOD : Word := 16#8207;   // Selected method is not supported
      ERR_REQUEST_SIZE : Word := 16#8210;   // Request array is too small for specified parameters
      ERR_RESPONSE_SIZE : Word := 16#8220;   // Receive buffer at parameter "responseData" too small
      ERR_CONN_LOST : Word := 16#8400;   // Offset for lost connection
      ERR_FORWARDING : Word := 16#8403;   // Server responded with forwarding message. Forwarding is not supported
      ERR_WEBSERVER : Word := 16#8404;   // Webserver responded with error code, see "diagnostics"
      ERR_INVALID_HEADER : Word := 16#8405;   // Header of response is invalid
      ERR_TIMEOUT : Word := 16#8408;   // Status: Time-out occurred
      ERR_UNDEFINED_STATE : Word := 16#8600;   // Status: Error due to an undefined state in state machine
      ERR_TSENDC : Word := 16#8601;   // Error: TCON encountered an error, see "diagnostics"
      ERR_TRCV : Word := 16#8603;   // Error: TURCV encountered error, see "diagnostics"
      ERR_MOVE_DATA_1 : Word := 16#8610;   // Error in MOVE_BLK_VARIANT to get length of data, see "diagnostics"
      ERR_MOVE_DATA_2 : Word := 16#8611;   // Error in MOVE_BLK_VARIANT to copy data, see "diagnostics"
      ERR_MOVE_USER_FIELDS : Word := 16#8612;   // Error in MOVE_BLK_VARIANT to copy user-defined header fields, see "diagnostics"
      ERR_ENCODING_UNKNOWN : Word := 16#8620;   // Transfer encoding of response could not be detected or is unsupported
      ERR_MOVE_IDENTITY : Word := 16#8630;   // Error in MOVE_BLK_VARIANT for transfer encoding 'identity', see "diagnostics"
      ERR_DECODING_FAILED : Word := 16#8640;   // Chunk encoded response could not be decoded
      ERR_MOVE_CHUNKED : Word := 16#8641;   // Error in MOVE_BLK_VARIANT for transfer encoding 'chunked', see "diagnostics"
      TSENDC_STATUS_CONNECTED : Word := 16#0001;   // TSEND_C: Communication connection established
      MOVE_STATUS_SIZE : Word := 16#8483;   // MOVE_BLK_VARIANT: DEST too small
      FB_STATE_NO_PROCESSING : USInt := 0;   // FB state: No processing
      FB_STATE_INIT : USInt := 1;   // FB state: initialization
      FB_STATE_REQUEST : USInt := 2;   // FB state: prepare request
      FB_STATE_SEND : USInt := 3;   // FB state: send request
      FB_STATE_RCV : USInt := 4;   // FB state: receive data
      FB_STATE_MON : USInt := 5;   // FB state: monitoring connection
      CRLF : String := '$R$L';   // Newline control character (carriage return, line feed)
      HEADER_END : String := '$R$L$R$L';   // End of HTTP header (two newline control characters)
      LEN_CRLF : UInt := 2;   // Length of CRLF
   END_VAR
   // statParam.paramIP.ConnPara.ActiveEstablished := true;
   // statParam.paramQDN.ConnPara.ActiveEstablished := true;
BEGIN
   REGION BLOCK INFO HEADER
     //===============================================================================
     // SIEMENS / (c)Copyright 2021
     //-------------------------------------------------------------------------------
     // Title:        LHTTP_PostPut
     // Function:     Implements the HTTP POST and PUT methods
     // Library:      LHTTP
     // Author:       Siemens Industry Online Support
     // Tested with:  CPU 1516-3 PN/DP V2.9
     // Engineering:  TIA Portal V17
     // Restrictions: --
     // Requirements: S7-1200 with firmware V4.4 or higher
     //               S7-1500 with firmware V2.0 or higher
     //-------------------------------------------------------------------------------
     // Change log table:
     // Version  | Date       | Expert in charge       | Changes applied
     //----------|------------|------------------------|------------------------------
     // 02.01.00 | 2021-12-15 | Online Support         | Added optional parameter "contentType" to make this header field adjustable
     //----------|------------|------------------------|------------------------------
     // 02.00.03 | 2021-05-10 | Online Support         | Fixed issues with chunked encoding
     //          |            |                        | Allow chunk sizes > 65535 Bytes
     //          |            |                        | Made header evaluation case-insensitive
     //----------|------------|------------------------|------------------------------
     // 02.00.00 | 2020-12-16 | Online Support         | Added support for PUT method
     //          |            |                        | Added option to keep connection established
     //          |            |                        | Added parameter to add user-defined headers fields
     //          |            |                        | Changed to data type of "data" to Variant to allow larger data
     //          |            |                        | Removed "statusID" and added "diagnostics" instead, changed some error codes
     //----------|------------|------------------------|------------------------------
     // 01.00.00 | 2019-04-01 | Online Support         | First released version
     //===============================================================================
   END_REGION

   REGION INSTRUCTIONS
     IF (#statStatus <> #STATUS_IDLE) THEN // Only execute when FB is triggered to reduce system load
       // Connect and send
       IF #statParam.isQDN THEN // Call if host is a domain name
         #instTSendC(REQ     := #statSend.req,
                     CONT    := #statSend.connect,
                     LEN     := #statRequest.length,
                     CONNECT := #statParam.paramQDN,
                     DATA    := #statRequest.chars);
       ELSE // Call if host is an IP address
         #instTSendC(REQ     := #statSend.req,
                     CONT    := #statSend.connect,
                     LEN     := #statRequest.length,
                     CONNECT := #statParam.paramIP,
                     DATA    := #statRequest.chars);
       END_IF;

       // Receive
       #instTRcv(ID    := #statParam.paramQDN.ConnPara.ID,
                 EN_R  := #statFBState >= #FB_STATE_RCV,
                 LEN   := 0,
                 ADHOC := true,
                 DATA  := #statRcvBuffer);

       // Monitor time out
       #instTimeout(IN := #statTimeoutIn,
                    PT := #timeOut);

       IF #instTimeout.Q THEN
         #statStatus := #ERR_TIMEOUT;
       END_IF;
     END_IF;
   END_REGION

   REGION TRIGGERING
     IF (#execute = true AND #statExecuteOld = false) // Check if FB is triggered
       AND (#statStatus = #STATUS_IDLE OR #statStatus = #STATUS_MONITORING)
     THEN // First call; initialize FB
       // Copy URL
       #tempUrl := #url;

       #statBusy := true;
       #statStatus := #STATUS_FIRST_CALL;
       #statSubfunctionStatus := #SUB_STATUS_NO_ERROR;
       #diagnostics := #statEmptyDiagnostics;

       IF #statConnected = FALSE THEN // Connection is not yet established
         #statFBState := #FB_STATE_INIT;
       ELSE // Connection is already established, skip init
         #statFBState := #FB_STATE_REQUEST;
       END_IF;

     ELSIF (#statStatus = #STATUS_FIRST_CALL) THEN
       #statStatus := #STATUS_CONNECTING;
     END_IF;

     // Edge detection 'execute' input
     #statExecuteOld := #execute;
   END_REGION TRIGGERING

   IF (#statStatus = #STATUS_IDLE) THEN // Nothing to do -> End here to reduce "system load"
     RETURN;
   END_IF;

   REGION STATE_MACHINE
     // State machine is wrapped in REPEAT loop to make it possible to quickly exit state machine
     // in case of an error or to go through CASE multiple times within one cycle
     REPEAT
       #tempExitLoop := true; // Condition to exit loop is set per default

       CASE #statFBState OF // State machine of FB
         #FB_STATE_NO_PROCESSING: // No processing active
           ;

         #FB_STATE_INIT:
           REGION INIT
             // Check data type of "data"
             IF TypeOf(#data) = String THEN
               #statDataIsString := TRUE;
             ELSIF TypeOfElements(#data) = Char THEN
               #statDataIsString := FALSE;
             ELSE
               #statStatus := #ERR_TYPE_DATA;
               EXIT;
             END_IF;

             // Get size of receive buffer
             IF LOWER_BOUND(ARR := #responseData, DIM := 1) <> 0 THEN
               #statStatus := #ERR_BOUND_NOT_ZERO;
               EXIT;
             ELSE
               #statSizeRcvArray := DINT_TO_UDINT(UPPER_BOUND(ARR := #responseData, DIM := 1)) + 1;
             END_IF;

             // Set connection parameters
             #statParam.paramQDN.ConnPara.InterfaceId := #hwID;
             #statParam.paramQDN.ConnPara.ID := #connID;
             #statParam.paramIP.ConnPara.InterfaceId := #hwID;
             #statParam.paramIP.ConnPara.ID := #connID;

             // Check if network protocol was specified to determine if connection should be secured
             #tempPos := FIND(IN1 := #tempUrl, IN2 := 'https://');
             IF #tempPos = 1 THEN // HTTPS
               #statParam.paramQDN.ActivateSecureConn := true;
               #statParam.paramQDN.ExtTLSCapabilities.%X0 := #tls.validateServerIdentity;
               #statParam.paramQDN.TLSServerCertRef := #tls.serverCert;
               #statParam.paramQDN.TLSClientCertRef := #tls.clientCert;
               #statParam.paramIP.ActivateSecureConn := true;
               #statParam.paramIP.ExtTLSCapabilities.%X0 := #tls.validateServerIdentity;
               #statParam.paramIP.TLSServerCertRef := #tls.serverCert;
               #statParam.paramIP.TLSClientCertRef := #tls.clientCert;
               // Delete network protocol from URL
               #tempUrl := DELETE(IN := #tempUrl, L := 8, P := 1);
             ELSE // HTTP
               #statParam.paramQDN.ActivateSecureConn := false;
               #statParam.paramIP.ActivateSecureConn := false;
               // Delete network protocol from URL if specified
               IF #tempUrl[5] = ':' THEN
                 #tempUrl := DELETE(IN := #tempUrl, L := 7, P := 1);
               END_IF;
             END_IF;

             // Determine if host is domain name or IP address
             #tempPos := CHAR_TO_INT(#tempUrl[1]);
             IF #tempPos >= CHAR_TO_INT('A') AND #tempPos <= CHAR_TO_INT('z') THEN // Host is a domain name
               #statParam.isQDN := true;
             ELSIF #tempPos >= CHAR_TO_INT('0') AND #tempPos <= CHAR_TO_INT('9') THEN // Host is an IP address
               #statParam.isQDN := false;
             ELSE // URL invalid
               #statStatus := #ERR_INVALID_URL;
               EXIT;
             END_IF;

             // Get host name and port
             #tempPos := FIND(IN1 := #tempUrl, IN2 := '/');
             IF #tempPos > 0 THEN // URL has a path after host name
               #statHost := LEFT(IN := #tempUrl, L := #tempPos - 1);
             ELSE
               #statHost := #tempUrl;
             END_IF;
             #tempPos := FIND(IN1 := #statHost, IN2 := ':');
             IF #tempPos > 0 THEN // Port specified in URL
               #statParam.paramQDN.ConnPara.RemotePort := STRING_TO_UINT(DELETE(IN := #statHost, L := #tempPos, P := 1));
               #statParam.paramIP.ConnPara.RemotePort := STRING_TO_UINT(DELETE(IN := #statHost, L := #tempPos, P := 1));
               #statHost := LEFT(IN := #statHost, L := #tempPos - 1);
             ELSE // No port specified in URL, set default port
               IF #statParam.paramQDN.ActivateSecureConn OR #statParam.paramIP.ActivateSecureConn THEN
                 #statParam.paramQDN.ConnPara.RemotePort := #PORT_SECURE;
                 #statParam.paramIP.ConnPara.RemotePort := #PORT_SECURE;
               ELSE
                 #statParam.paramQDN.ConnPara.RemotePort := #PORT_UNSECURE;
                 #statParam.paramIP.ConnPara.RemotePort := #PORT_UNSECURE;
               END_IF;
             END_IF;

             IF #statParam.isQDN THEN // Host is a domain name
               #statParam.paramQDN.ConnPara.RemoteQDN := CONCAT(IN1 := #statHost, IN2 := '.');
             ELSE // Host is an IP address
               #tempString := #statHost;
               FOR #tempIndex := 1 TO 3 DO
                 #tempPos := FIND(IN1 := #tempString, IN2 := '.');
                 #statParam.paramIP.ConnPara.RemoteAddress.ADDR[#tempIndex] := UINT_TO_BYTE(STRING_TO_UINT(LEFT(IN := #tempString, L := #tempPos - 1)));
                 #tempString := DELETE(IN := #tempString, L := #tempPos, P := 1);
               END_FOR;
               #statParam.paramIP.ConnPara.RemoteAddress.ADDR[4] := UINT_TO_BYTE(STRING_TO_UINT(#tempString));
             END_IF;

             #statFBState := #FB_STATE_REQUEST;
             #tempExitLoop := FALSE; // Don't exit loop to go directly to prepare request
           END_REGION INIT

         #FB_STATE_REQUEST:
           REGION PREP_REQUEST
             // Get content length
             // Content length is evaluated first so that request array can be used for this to save memory
             IF #statDataIsString THEN
               VariantGet(SRC := #data,
                          DST => #tempData);
               #tempLenData := INT_TO_UINT(LEN(#tempData));
             ELSE // "data" is Array of Char
               #tempLen := UDINT_TO_UINT(CountOfElements(#data));
               #tempRet := INT_TO_WORD(MOVE_BLK_VARIANT(SRC := #data, COUNT := #tempLen, SRC_INDEX := 0, DEST_INDEX := 0, DEST => #statRequest.chars));

               IF #tempRet = #MOVE_STATUS_SIZE THEN
                 #statStatus := #ERR_REQUEST_SIZE;
                 EXIT;
               ELSIF #tempRet <> 16#0000 THEN
                 #statStatus := #ERR_MOVE_DATA_1;
                 #statSubfunctionStatus := #tempRet;
                 EXIT;
               END_IF;

               FOR #tempIndex := 0 TO UINT_TO_DINT(#tempLen) DO
                 IF #statRequest.chars[#tempIndex] = '$00' THEN
                   #tempLenData := DINT_TO_UINT(#tempIndex);
                   EXIT;
                 END_IF;
               END_FOR;

               IF #tempLenData = 0 THEN
                 #statStatus := #ERR_END_DATA;
                 EXIT;
               END_IF;
             END_IF;

             // Set method
             IF #method = #METHOD_POST THEN
               #tempString := 'POST ';
             ELSIF #method = #METHOD_PUT THEN
               #tempString := 'PUT ';
             ELSE
               #statStatus := #ERR_METHOD;
               EXIT;
             END_IF;

             // Check host in URL when using existing connection
             IF #statConnected = TRUE THEN
               #tempPos := FIND(IN1 := #tempUrl, IN2 := #statHost);
               IF #tempPos = 0 THEN // URL doesn't contain expected host
                 #statStatus := #ERR_DIFFERENT_HOST;
                 EXIT;
               ELSE // Scheme and host must be deleted for further processing
                 #tempUrl := DELETE(IN := #tempUrl, L := #tempPos + LEN(#statHost) - 1, P := 1);
               END_IF;
             END_IF;

             // Get path
             #tempPos := FIND(IN1 := #tempUrl, IN2 := '/');
             IF #tempPos > 0 THEN // URL has a path after host name
               #tempPath := DELETE(IN := #tempUrl, L := #tempPos - 1, P := 1);
             ELSE
               #tempPath := '/';
             END_IF;

             // Put together request
             // Strg_TO_Chars conversion is done several times to utilize maximum length of parameter url
             Strg_TO_Chars(Strg   := CONCAT(IN1 := #tempString, IN2 := #tempPath), // Path cannot be longer than 249 characters --> save to use CONCAT
                           pChars := 0,
                           Cnt    => #tempLen,
                           Chars  := #statRequest.chars);
             #tempPos := UINT_TO_INT(#tempLen);

             Strg_TO_Chars(Strg   := CONCAT(IN1 := ' HTTP/1.1$R$LHost: ', IN2 := #statHost), // Host will not use all 254 characters --> save to use CONCAT
                           pChars := #tempPos,
                           Cnt    => #tempLen,
                           Chars  := #statRequest.chars);
             #tempPos += UINT_TO_INT(#tempLen);

             Strg_TO_Chars(Strg   := '$R$LUser-Agent: SIMATIC Controller (LHTTP)$R$LConnection: keep-alive$R$LAccept-Charset: utf-8$R$LContent-Encoding: identity$R$L',
                           pChars := #tempPos,
                           Cnt    => #tempLen,
                           Chars  := #statRequest.chars);
             #tempPos += UINT_TO_INT(#tempLen);

             Strg_TO_Chars(Strg   := CONCAT(IN1 := 'Content-Type: ', IN2 := #contentType, IN3 := '$R$L'),
                           pChars := #tempPos,
                           Cnt    => #tempLen,
                           Chars  := #statRequest.chars);
             #tempPos += UINT_TO_INT(#tempLen);

             Strg_TO_Chars(Strg   := CONCAT(IN1 := 'Content-Length: ', IN2 := DELETE(IN := UINT_TO_STRING(#tempLenData), L := 1, P := 1), IN3 := #CRLF),
                           pChars := #tempPos,
                           Cnt    => #tempLen,
                           Chars  := #statRequest.chars);
             #tempPos += UINT_TO_INT(#tempLen);

             // Insert additional user-defined header fields
             IF #userFields[0] <> ' ' THEN
               FOR #tempLen := 0 TO #UPPER_USER_FIELDS DO
                 IF #userFields[#tempLen] = '$00' THEN
                   EXIT;
                 END_IF;
               END_FOR;

               IF #tempLen > #UPPER_USER_FIELDS THEN // End not found
                 #statStatus := #ERR_END_USER_FIELDS;
                 EXIT;
               END_IF;

               #tempRet := INT_TO_WORD(MOVE_BLK_VARIANT(SRC := #userFields, COUNT := #tempLen, SRC_INDEX := 0, DEST_INDEX := #tempPos, DEST => #statRequest.chars));

               IF #tempRet = #MOVE_STATUS_SIZE THEN
                 #statStatus := #ERR_REQUEST_SIZE;
                 EXIT;
               ELSIF #tempRet <> 16#0000 THEN
                 #statStatus := #ERR_MOVE_USER_FIELDS;
                 #statSubfunctionStatus := #tempRet;
                 EXIT;
               END_IF;

               #tempPos += UINT_TO_INT(#tempLen);

               // Append CRLF if needed
               IF #statRequest.chars[#tempPos - 2] <> '$R' AND #statRequest.chars[#tempPos - 1] <> '$L' THEN
                 #statRequest.chars[#tempPos] := '$R';
                 #statRequest.chars[#tempPos + 1] := '$L';
                 #tempPos += 2;
               END_IF;
             END_IF;

             // Append end of header section
             Strg_TO_Chars(Strg   := #CRLF,
                           pChars := #tempPos,
                           Cnt    => #tempLen,
                           Chars  := #statRequest.chars);
             #tempPos += UINT_TO_INT(#tempLen);

             // Append data
             IF TypeOf(#data) = String THEN
               Strg_TO_Chars(Strg   := #tempData,
                             pChars := #tempPos,
                             Cnt    => #tempLenData,
                             Chars  := #statRequest.chars);
             ELSE // "data" is Array of Char
               #tempRet := INT_TO_WORD(MOVE_BLK_VARIANT(SRC := #data, COUNT := #tempLenData, SRC_INDEX := 0, DEST_INDEX := #tempPos, DEST => #statRequest.chars));

               IF #tempRet = #MOVE_STATUS_SIZE THEN
                 #statStatus := #ERR_REQUEST_SIZE;
                 EXIT;
               ELSIF #tempRet <> 16#0000 THEN
                 #statStatus := #ERR_MOVE_DATA_2;
                 #statSubfunctionStatus := #tempRet;
                 EXIT;
               END_IF;
             END_IF;

             // Calculate total length of request
             #statRequest.length := INT_TO_UINT(#tempPos) + #tempLenData;

             #statSend.connect := true; // Connect
             #statSend.req := true; // Send request
             #statTimeoutIn := true; // Start timer
             #statFBState := #FB_STATE_SEND;
           END_REGION

         #FB_STATE_SEND: // Send data
           REGION SEND
             IF #instTSendC.STATUS = #TSENDC_STATUS_CONNECTED THEN
               #statConnected := TRUE;
             ELSIF #instTSendC.DONE THEN
               #statStatus := #STATUS_SENT;
               #statFBState := #FB_STATE_RCV;
               // Don't exit loop to go directly to receive state
               // without waiting for next cycle so that no responses can be missed
               #tempExitLoop := false;
             ELSIF #instTSendC.ERROR THEN
               #statStatus := #ERR_TSENDC;
               #statSubfunctionStatus := #instTSendC.STATUS;
             END_IF;
           END_REGION

         #FB_STATE_RCV: // Wait for new data
           REGION RCV
             IF #instTRcv.NDR THEN

               REGION HEADER_EVAL
                 // Evaluate header if received packet is first packet
                 IF #statEncoding = '' THEN
                   // Get response code
                   Chars_TO_Strg(Chars  := #statRcvBuffer,
                                 pChars := #POS_RESPONSE_CODE,
                                 Cnt    := 3,
                                 Strg   => #tempString);
                   #statResponseCode := STRING_TO_UINT(#tempString);

                   // Exit loop immediately and output errror if response code shows errors or forwarding
                   IF #statResponseCode >= 300 THEN
                     #tempRet := ATH(IN := #tempString, N := 3, OUT => #statSubfunctionStatus); // Interpret response code as hexadecimal
                     #statSubfunctionStatus := SHR(IN := #statSubfunctionStatus, N := 20);
                     IF #statResponseCode >= 400 THEN
                       #statStatus := #ERR_WEBSERVER;
                     ELSE
                       #statStatus := #ERR_FORWARDING;
                     END_IF;
                     EXIT;
                   END_IF;

                   // Get length of HTTP header
                   #tempLen := DINT_TO_UINT("LHTTP_FindStringInArray"(searchFor := #HEADER_END, searchIn := #statRcvBuffer) + LEN(#HEADER_END));

                   // Exit loop immediately and output errror if header end cannot be found
                   IF #tempLen = 0 THEN
                     #statStatus := #ERR_INVALID_HEADER;
                     EXIT;
                   END_IF;

                   // Search header for content length
                   #tempRet := "LHTTP_ExtractStringFromArray"(textBefore := 'Content-Length: ',
                                                              textAfter := #CRLF,
                                                              extractedString => #tempString,
                                                              searchIn := #statRcvBuffer);

                   IF #tempRet <> 0 THEN // Content length not found; try lower-case
                     #tempRet := "LHTTP_ExtractStringFromArray"(textBefore := 'content-length: ',
                                                                textAfter := #CRLF,
                                                                extractedString => #tempString,
                                                                searchIn := #statRcvBuffer);
                   END_IF;

                   IF #tempRet = 0 THEN // Content length found
                     #statContentLength := STRING_TO_UINT(#tempString);
                     #statEncoding := 'identity';
                   ELSE // Can't detect content length, check if transfer encoding is 'chunked'
                     #tempPos := DINT_TO_INT("LHTTP_FindStringInArray"(searchFor := 'chunked', searchIn := #statRcvBuffer));

                     IF #tempPos >= 0 THEN
                       #statEncoding := 'chunked';
                     ELSE // Exit loop immediately and output error if content length nor transfer encoding can be detected
                       #statStatus := #ERR_ENCODING_UNKNOWN;
                       EXIT;
                     END_IF;
                   END_IF;

                   IF #instTRcv.RCVD_LEN = #tempLen THEN // Packet contains no body, wait for next packet
                     EXIT;
                   END_IF;
                 END_IF;
               END_REGION

               REGION TE_IDENTITY
                 IF #statEncoding = 'identity' THEN // Transfer encoding is 'identity'
                   // Move data from buffer to output; tempLen contains header length during first packet, otherwise 0
                   #tempRet := INT_TO_WORD(MOVE_BLK_VARIANT(SRC := #statRcvBuffer,
                                                                                    COUNT := MIN(IN1 := #instTRcv.RCVD_LEN - #tempLen, IN2 := #statSizeRcvArray - #statRcvdLen), // Move as much as possible to output
                                                                                    SRC_INDEX := #tempLen,
                                                                                    DEST_INDEX := UDINT_TO_DINT(#statRcvdLen),
                                                                                    DEST => #responseData));

                   // Exit loop immediately and output error if data could not be moved
                   IF #tempRet <> 0 THEN
                     #statStatus := #ERR_MOVE_IDENTITY;
                     #statSubfunctionStatus := #tempRet;
                     EXIT;
                   END_IF;

                   // Add length of received packet to sum; tempLen contains header length during first packet, otherwise 0
                   #statRcvdLen += #instTRcv.RCVD_LEN - #tempLen;

                   IF #statRcvdLen > #statSizeRcvArray THEN // Receive buffer too small
                     #statStatus := #ERR_RESPONSE_SIZE;
                     #statLength := #statContentLength; // Output required size of buffer
                   ELSIF #statRcvdLen >= #statContentLength THEN // Everything was received
                     #statStatus := #STATUS_DONE;
                     #statLength := #statRcvdLen;
                   END_IF;
                 END_IF;
               END_REGION

               REGION TE_CHUNKED
                 IF #statEncoding = 'chunked' THEN // Transfer encoding is 'chunked'

                   // Set position of chunk data
                   #tempChunk.posData := #tempLen; // tempLen contains header length during first packet, otherwise 0

                   REPEAT
                     #tempChunk.exitLoop := true; // Condition to exit loop is set per default

                     // Read length of chunk if received packet is first packet or a previous chunk was received completely
                     IF #statChunkLen = 0 THEN
                       // Extract hexadecimal chunk-size field
                       Chars_TO_Strg(Chars  := #statRcvBuffer,
                                     pChars := #tempChunk.posData,
                                     Cnt    := 0,
                                     Strg   => #tempString);
                       #tempPos := FIND(IN1 := #tempString, IN2 := #CRLF);
                       #tempRet := ATH(IN := #tempString, N := #tempPos - 1, OUT => #statChunkLen);
                       // Shift bits to the right depending on length of chunk size, since ATH is left aligned
                       #statChunkLen := SHR(IN := #statChunkLen, N := 4 * INT_TO_UINT(8 - (#tempPos - 1)));

                       // Move start position of data behind chunk-size field
                       #tempChunk.posData += INT_TO_UINT(#tempPos) + 1;

                       // Exit loop immediately and output error if chunk size cannot be detected
                       IF #tempRet <> 0 THEN
                         #statStatus := #ERR_DECODING_FAILED;
                         EXIT;
                       END_IF;
                     END_IF;

                     IF #statChunkLen = 0 THEN // Length was evaluated, chunk contains no data --> final chunk received
                       #statStatus := #STATUS_DONE;
                       #statLength := #statRcvdLen;
                     ELSE // Chunk contains data
                       // Evaluate length of received packet and set length of data accordingly
                       IF #instTRcv.RCVD_LEN = #tempChunk.posData + #statChunkLen + #LEN_CRLF THEN // Chunk was received entirely and packet contains no further chunks
                         #tempChunk.lenData := UDINT_TO_UINT(#statChunkLen); // Output remaining length of chunk
                       ELSIF #instTRcv.RCVD_LEN < #tempChunk.posData + #statChunkLen + #LEN_CRLF THEN // Packet only contains part of chunk
                         #tempChunk.lenData := UDINT_TO_UINT(#instTRcv.RCVD_LEN) - #tempChunk.posData; // Output entire packet without possible chunk-size field
                       ELSIF #instTRcv.RCVD_LEN > #tempChunk.posData + #statChunkLen + #LEN_CRLF THEN // Current packet contains more than one chunk
                         #tempChunk.lenData := UDINT_TO_UINT(#statChunkLen); // Output remaining length of chunk
                         #tempChunk.exitLoop := false; // Execute loop again since packet contains more data
                       ELSE // Can't decode message
                         #statStatus := #ERR_DECODING_FAILED;
                         EXIT;
                       END_IF;

                       // Move received data to output
                       #tempRet := INT_TO_WORD(MOVE_BLK_VARIANT(SRC := #statRcvBuffer,
                                                                                        COUNT := MIN(IN1 := #tempChunk.lenData, IN2 := #statSizeRcvArray - #statRcvdLen), // Move as much as possible to output
                                                                                        SRC_INDEX := #tempChunk.posData,
                                                                                        DEST_INDEX := UDINT_TO_DINT(#statRcvdLen),
                                                                                        DEST => #responseData));

                       // Exit loop immediately and output error if data could not be moved
                       IF #tempRet <> 0 THEN
                         #statStatus := #ERR_MOVE_CHUNKED;
                         #statSubfunctionStatus := #tempRet;
                         EXIT;
                       END_IF;

                       // Move start position of data behind data of current chunk in case packet contains more data; only relevant if REPEAT loop is executed again
                       #tempChunk.posData += #tempChunk.lenData + #LEN_CRLF;

                       // Subtract length of data in current packet from remaining length of chunk and add to sum of received data
                       #statChunkLen -= #tempChunk.lenData;
                       #statRcvdLen += #tempChunk.lenData;

                       IF #statRcvdLen > #statSizeRcvArray THEN // Receive buffer too small
                         #statStatus := #ERR_RESPONSE_SIZE;
                         #statLength := #statRcvdLen; // Output required size of buffer according to so far received chunked messages
                         EXIT;
                       END_IF;
                     END_IF;
                   UNTIL (#tempChunk.exitLoop = true) END_REPEAT;
                 END_IF;
               END_REGION

             ELSIF #instTRcv.ERROR THEN
               #statStatus := #ERR_TRCV;
               #statSubfunctionStatus := #instTRcv.STATUS;
             END_IF;
           END_REGION

         #FB_STATE_MON:
           REGION MONITORING
             IF #keepConnection = FALSE THEN // Trigger to disconnect
               #statSend.connect := FALSE;
               #statDone := FALSE;
               #statBusy := TRUE;
               #statStatus := #STATUS_DISCONNECTING;
             END_IF;

             IF #instTSendC.STATUS = #STATUS_DISCONNECTED THEN
               #statConnected := FALSE;
               #statStatus := #STATUS_DISCONNECTED;
             ELSIF #instTRcv.ERROR THEN
               #statConnected := FALSE;
               #statStatus := #ERR_CONN_LOST OR (#instTRcv.STATUS AND 16#00FF);
             END_IF;
           END_REGION

         ELSE // Undefined state in state machine reached
           #statStatus := #ERR_UNDEFINED_STATE;
       END_CASE;

     UNTIL (#tempExitLoop = true) END_REPEAT;
   END_REGION

   REGION OUTPUTS
     // Write outputs
     IF (#statStatus = #STATUS_DONE) AND (#statDone = false) THEN // Execution finished without errors
       #statDone := true;
       #statBusy := false;
       #statError := false;
       #statSend.connect := #keepConnection;
       #statSend.req := false;
       #statTimeoutIn := false;

       IF #keepConnection THEN
         // execution finished but connection is kept alive --> set state monitoring
         #statFBState := #FB_STATE_MON;
       ELSE
         #statConnected := FALSE;
         // execution finished --> set state no processing
         #statFBState := #FB_STATE_NO_PROCESSING;
       END_IF;

     ELSIF (#statStatus = #STATUS_DISCONNECTED) AND (#statBusy = true) THEN // Connection was terminated separately of send job
       #statConnected := FALSE;
       #statBusy := FALSE;
       // execution finished --> set state no processing
       #statFBState := #FB_STATE_NO_PROCESSING;

     ELSIF (#statStatus.%X15 = true) AND (#statError = false) THEN // Error occurred (#statStatus is 16#8000 to 16#FFFF)
       #statConnected := false;
       #statDone := false;
       #statBusy := false;
       #statError := true;
       #statSend.connect := false; // After error, connection is always terminated
       #statSend.req := false;
       #statTimeoutIn := false;
       // Write diagnostics
       #diagnostics.status := #statStatus;
       #diagnostics.subfunctionStatus := #statSubfunctionStatus;
       #diagnostics.stateNumber := #statFBState;
       // execution aborted --> set state no processing
       #statFBState := #FB_STATE_NO_PROCESSING;

     ELSIF ((#execute = false) AND ((#statDone = true) OR (#statError = true)))
       OR ((#statStatus = #STATUS_DISCONNECTED) AND (#statBusy = false)) // Connection was terminated separately of send job
     THEN // Reset outputs
       #statDone := false;
       #statBusy := false;
       #statError := false;
       #statResponseCode := 0;
       #statLength := 0;
       #statContentLength := 0;
       #statChunkLen := 0;
       #statEncoding := '';
       #statRcvdLen := 0;

       IF #statConnected THEN
         #statStatus := #STATUS_MONITORING;
       ELSE
         #statStatus := #STATUS_IDLE;
       END_IF;
     END_IF;

     // Write static values to outputs
     #connected := #statConnected;
     #done := #statDone;
     #busy := #statBusy;
     #error := #statError;
     #status := #statStatus;
     #responseCode := #statResponseCode;
     #length := #statLength;
     ENO := NOT #statError;
   END_REGION OUTPUTS
END_FUNCTION_BLOCK

// folder: 1000_HTTP/LHTTP/Utilities

